LIN {X 0,Y 250.875,Z 1142.399,A -85,B 0,C 180,E1 12020.082,E2 12020.082} C_VEL
LIN {X 0,Y 256.452,Z 1121.884,A -85,B 0,C 180,E1 12017.28,E2 12017.28} C_VEL
LIN {X 0,Y 262.071,Z 1099.557,A -85,B 0,C 180,E1 12014.793,E2 12014.793} C_VEL
LIN {X 0,Y 267.365,Z 1075.91,A -85,B 0,C 180,E1 12012.685,E2 12012.685} C_VEL
LIN {X 0,Y 272.115,Z 1051.396,A -85,B 0,C 180,E1 12010.964,E2 12010.964} C_VEL
LIN {X 0,Y 276.224,Z 1025.533,A -85,B 0,C 180,E1 12009.582,E2 12009.582} C_VEL
LIN {X 0,Y 282.995,Z 970.684,A -85,B 0,C 180,E1 12007.498,E2 12007.498} C_VEL
LIN {X 0,Y 300.587,Z 832.085,A -85,B 0,C 180,E1 12002.78,E2 12002.78} C_VEL
LIN {X 0,Y 288.306,Z 807.074,A -85,B 0,C 180,E1 11999.364,E2 11999.364} C_VEL
LIN {X 0,Y 276.041,Z 783.888,A -85,B 0,C 180,E1 11995.652,E2 11995.652} C_VEL
LIN {X 0,Y 264.408,Z 763.41,A -85,B 0,C 180,E1 11991.784,E2 11991.784} C_VEL
LIN {X 0,Y 253.537,Z 745.664,A -85,B 0,C 180,E1 11987.8,E2 11987.8} C_VEL
LIN {X 0,Y 245.018,Z 732.558,A -85,B 0,C 180,E1 11984.357,E2 11984.357} C_VEL
LIN {X 0,Y 243.38,Z 730.234,A -85,B 0,C 180,E1 11983.667,E2 11983.667} C_VEL
LIN {X 0,Y 242.49,Z 729.861,A -85,B 0,C 180,E1 11983.311,E2 11983.311} C_VEL
LIN {X 0,Y 243.74,Z 731.685,A -85,B 0,C 180,E1 11981.348,E2 11981.348} C_VEL
LIN {X 0,Y 246.278,Z 736.647,A -85,B 0,C 180,E1 11977.233,E2 11977.233} C_VEL
LIN {X 0,Y 248.775,Z 741.662,A -85,B 0,C 180,E1 11973.69,E2 11973.69} C_VEL
LIN {X 0,Y 251.092,Z 746.409,A -85,B 0,C 180,E1 11970.688,E2 11970.688} C_VEL
LIN {X 0,Y 254.649,Z 753.588,A -85,B 0,C 180,E1 11966.627,E2 11966.627} C_VEL
LIN {X 0,Y 258.733,Z 762.816,A -85,B 0,C 180,E1 11962.23,E2 11962.23} C_VEL
LIN {X 0,Y 263.13,Z 773.088,A -85,B 0,C 180,E1 11957.94,E2 11957.94} C_VEL
LIN {X 0,Y 267.756,Z 784.772,A -85,B 0,C 180,E1 11953.685,E2 11953.685} C_VEL
LIN {X 0,Y 272.379,Z 797.535,A -85,B 0,C 180,E1 11949.593,E2 11949.593} C_VEL
LIN {X 0,Y 277.126,Z 811.99,A -85,B 0,C 180,E1 11945.489,E2 11945.489} C_VEL
LIN {X 0,Y 281.607,Z 827.392,A -85,B 0,C 180,E1 11941.593,E2 11941.593} C_VEL
LIN {X 0,Y 283.554,Z 835.371,A -85,B 0,C 180,E1 11939.762,E2 11939.762} C_VEL
LIN {X 0,Y 271.947,Z 876.824,A -85,B 0,C 180,E1 11934.348,E2 11934.348} C_VEL
LIN {X 0,Y 261.07,Z 920.048,A -85,B 0,C 180,E1 11928.508,E2 11928.508} C_VEL
LIN {X 0,Y 258.223,Z 932.884,A -85,B 0,C 180,E1 11926.79,E2 11926.79} C_VEL
LIN {X 0,Y 257.872,Z 942.975,A -85,B 0,C 180,E1 11926.225,E2 11926.225} C_VEL
LIN {X 0,Y 250.822,Z 1001.369,A -85,B 0,C 180,E1 11923.289,E2 11923.289} C_VEL
LIN {X 0,Y 244.667,Z 1051.459,A -85,B 0,C 180,E1 11920.196,E2 11920.196} C_VEL
LIN {X 0,Y 240.696,Z 1089.833,A -85,B 0,C 180,E1 11917.338,E2 11917.338} C_VEL
LIN {X 0,Y 238.457,Z 1107.896,A -85,B 0,C 180,E1 11915.523,E2 11915.523} C_VEL
LIN {X 0,Y 236.095,Z 1124.174,A -85,B 0,C 180,E1 11913.406,E2 11913.406} C_VEL
LIN {X 0,Y 233.562,Z 1140.25,A -85,B 0,C 180,E1 11910.77,E2 11910.77} C_VEL
LIN {X 0,Y 231.041,Z 1155.81,A -85,B 0,C 180,E1 11907.586,E2 11907.586} C_VEL
LIN {X 0,Y 228.852,Z 1169.954,A -85,B 0,C 180,E1 11903.975,E2 11903.975} C_VEL
LIN {X 0,Y 227.359,Z 1181.506,A -85,B 0,C 180,E1 11900.33,E2 11900.33} C_VEL
LIN {X 0,Y 226.431,Z 1192.191,A -85,B 0,C 180,E1 11896.153,E2 11896.153} C_VEL
LIN {X 0,Y 226.295,Z 1201.142,A -85,B 0,C 180,E1 11891.727,E2 11891.727} C_VEL
LIN {X 0,Y 227.021,Z 1207.997,A -85,B 0,C 180,E1 11887.338,E2 11887.338} C_VEL
LIN {X 0,Y 228.861,Z 1213.356,A -85,B 0,C 180,E1 11882.755,E2 11882.755} C_VEL
LIN {X 0,Y 232.16,Z 1217.018,A -85,B 0,C 180,E1 11878.025,E2 11878.025} C_VEL
LIN {X 0,Y 236.961,Z 1218.837,A -85,B 0,C 180,E1 11873.458,E2 11873.458} C_VEL
LIN {X 0,Y 243.636,Z 1218.792,A -85,B 0,C 180,E1 11868.878,E2 11868.878} C_VEL
LIN {X 0,Y 252.162,Z 1216.676,A -85,B 0,C 180,E1 11864.47,E2 11864.47} C_VEL
LIN {X 0,Y 261.202,Z 1213.007,A -85,B 0,C 180,E1 11860.779,E2 11860.779} C_VEL
LIN {X 0,Y 271.771,Z 1207.47,A -85,B 0,C 180,E1 11857.275,E2 11857.275} C_VEL
LIN {X 0,Y 283.551,Z 1200.008,A -85,B 0,C 180,E1 11854.07,E2 11854.07} C_VEL
LIN {X 0,Y 286.866,Z 1197.645,A -85,B 0,C 180,E1 11853.267,E2 11853.267} C_VEL
LIN {X 0,Y 290.92,Z 1194.738,A -85,B 0,C 180,E1 11852.083,E2 11852.083} C_VEL
LIN {X 0,Y 299.595,Z 1187.805,A -85,B 0,C 180,E1 11848.837,E2 11848.837} C_VEL
LIN {X 0,Y 303.94,Z 1184.184,A -85,B 0,C 180,E1 11847.843,E2 11847.843} C_VEL
LIN {X 0,Y 312.8,Z 1176.577,A -85,B 0,C 180,E1 11846.411,E2 11846.411} C_VEL
LIN {X 0,Y 298.241,Z 1190.287,A -85,B 0,C 180,E1 11844.221,E2 11844.221} C_VEL
LIN {X 0,Y 282.111,Z 1204.39,A -85,B 0,C 180,E1 11841.232,E2 11841.232} C_VEL
LIN {X 0,Y 267.332,Z 1216.538,A -85,B 0,C 180,E1 11837.775,E2 11837.775} C_VEL
LIN {X 0,Y 252.966,Z 1227.89,A -85,B 0,C 180,E1 11833.448,E2 11833.448} C_VEL
LIN {X 0,Y 240.286,Z 1237.665,A -85,B 0,C 180,E1 11828.313,E2 11828.313} C_VEL
LIN {X 0,Y 230.902,Z 1244.993,A -85,B 0,C 180,E1 11823.063,E2 11823.063} C_VEL
LIN {X 0,Y 223.215,Z 1251.335,A -85,B 0,C 180,E1 11816.608,E2 11816.608} C_VEL
LIN {X 0,Y 218.765,Z 1255.587,A -85,B 0,C 180,E1 11809.687,E2 11809.687} C_VEL
LIN {X 0,Y 217.644,Z 1257.45,A -85,B 0,C 180,E1 11804.496,E2 11804.496} C_VEL
LIN {X 0,Y 217.156,Z 1265.482,A -85,B 0,C 180,E1 11799.805,E2 11799.805} C_VEL
LIN {X 0,Y 217.229,Z 1272.099,A -85,B 0,C 180,E1 11795.014,E2 11795.014} C_VEL
LIN {X 0,Y 217.292,Z 1276.222,A -85,B 0,C 180,E1 11791.051,E2 11791.051} C_VEL
LIN {X 0,Y 217,Z 1279.073,A -85,B 0,C 180,E1 11787.355,E2 11787.355} C_VEL
LIN {X 0,Y 216.544,Z 1281.409,A -85,B 0,C 180,E1 11782.835,E2 11782.835} C_VEL
LIN {X 0,Y 216.902,Z 1282.929,A -85,B 0,C 180,E1 11776.578,E2 11776.578} C_VEL
LIN {X 0,Y 219.361,Z 1282.777,A -85,B 0,C 180,E1 11770.284,E2 11770.284} C_VEL
LIN {X 0,Y 224.928,Z 1280.78,A -85,B 0,C 180,E1 11763.603,E2 11763.603} C_VEL
LIN {X 0,Y 234.376,Z 1276.835,A -85,B 0,C 180,E1 11756.899,E2 11756.899} C_VEL
LIN {X 0,Y 246.727,Z 1271.422,A -85,B 0,C 180,E1 11751.083,E2 11751.083} C_VEL
LIN {X 0,Y 263.196,Z 1263.992,A -85,B 0,C 180,E1 11745.648,E2 11745.648} C_VEL
LIN {X 0,Y 272.977,Z 1259.532,A -85,B 0,C 180,E1 11743.089,E2 11743.089} C_VEL
LIN {X 0,Y 255.858,Z 1264.797,A -85,B 0,C 180,E1 11738.131,E2 11738.131} C_VEL
LIN {X 0,Y 241.819,Z 1268.371,A -85,B 0,C 180,E1 11732.516,E2 11732.516} C_VEL
LIN {X 0,Y 231.077,Z 1270.191,A -85,B 0,C 180,E1 11726.395,E2 11726.395} C_VEL
LIN {X 0,Y 223.504,Z 1270.13,A -85,B 0,C 180,E1 11719.877,E2 11719.877} C_VEL
LIN {X 0,Y 219.062,Z 1268.343,A -85,B 0,C 180,E1 11713.461,E2 11713.461} C_VEL
LIN {X 0,Y 216.939,Z 1264.947,A -85,B 0,C 180,E1 11707.149,E2 11707.149} C_VEL
LIN {X 0,Y 216.319,Z 1260.682,A -85,B 0,C 180,E1 11701.854,E2 11701.854} C_VEL
LIN {X 0,Y 216.214,Z 1255.219,A -85,B 0,C 180,E1 11696.819,E2 11696.819} C_VEL
LIN {X 0,Y 216.471,Z 1248.644,A -85,B 0,C 180,E1 11692.035,E2 11692.035} C_VEL
LIN {X 0,Y 217.315,Z 1239.961,A -85,B 0,C 180,E1 11686.97,E2 11686.97} C_VEL
LIN {X 0,Y 218.948,Z 1230.048,A -85,B 0,C 180,E1 11682.183,E2 11682.183} C_VEL
LIN {X 0,Y 221.732,Z 1217.438,A -85,B 0,C 180,E1 11677.181,E2 11677.181} C_VEL
LIN {X 0,Y 225.229,Z 1204.04,A -85,B 0,C 180,E1 11672.789,E2 11672.789} C_VEL
LIN {X 0,Y 229.707,Z 1188.379,A -85,B 0,C 180,E1 11668.51,E2 11668.51} C_VEL
LIN {X 0,Y 235.034,Z 1170.475,A -85,B 0,C 180,E1 11664.468,E2 11664.468} C_VEL
LIN {X 0,Y 240.517,Z 1152.019,A -85,B 0,C 180,E1 11661.028,E2 11661.028} C_VEL
LIN {X 0,Y 246.057,Z 1132.723,A -85,B 0,C 180,E1 11658.047,E2 11658.047} C_VEL
LIN {X 0,Y 251.937,Z 1110.749,A -85,B 0,C 180,E1 11655.272,E2 11655.272} C_VEL
LIN {X 0,Y 257.513,Z 1087.985,A -85,B 0,C 180,E1 11652.952,E2 11652.952} C_VEL
LIN {X 0,Y 262.772,Z 1063.42,A -85,B 0,C 180,E1 11650.963,E2 11650.963} C_VEL
LIN {X 0,Y 267.339,Z 1038.17,A -85,B 0,C 180,E1 11649.382,E2 11649.382} C_VEL
LIN {X 0,Y 271.084,Z 1012.485,A -85,B 0,C 180,E1 11648.187,E2 11648.187} C_VEL
LIN {X 0,Y 294.09,Z 834.845,A -85,B 0,C 180,E1 11641.891,E2 11641.891} C_VEL
LIN {X 0,Y 282.266,Z 810.63,A -85,B 0,C 180,E1 11638.485,E2 11638.485} C_VEL
LIN {X 0,Y 269.829,Z 787,A -85,B 0,C 180,E1 11634.582,E2 11634.582} C_VEL
LIN {X 0,Y 258.588,Z 767.172,A -85,B 0,C 180,E1 11630.694,E2 11630.694} C_VEL
LIN {X 0,Y 248.246,Z 750.166,A -85,B 0,C 180,E1 11626.741,E2 11626.741} C_VEL
LIN {X 0,Y 240.071,Z 737.582,A -85,B 0,C 180,E1 11623.307,E2 11623.307} C_VEL
LIN {X 0,Y 238.286,Z 736.957,A -85,B 0,C 180,E1 11622.668,E2 11622.668} C_VEL
LIN {X 0,Y 239.049,Z 738.368,A -85,B 0,C 180,E1 11621.341,E2 11621.341} C_VEL
LIN {X 0,Y 241.442,Z 743.073,A -85,B 0,C 180,E1 11617.379,E2 11617.379} C_VEL
LIN {X 0,Y 243.73,Z 747.729,A -85,B 0,C 180,E1 11614.002,E2 11614.002} C_VEL
LIN {X 0,Y 246.014,Z 752.518,A -85,B 0,C 180,E1 11610.935,E2 11610.935} C_VEL
LIN {X 0,Y 249.344,Z 759.346,A -85,B 0,C 180,E1 11607.015,E2 11607.015} C_VEL
LIN {X 0,Y 253.36,Z 768.616,A -85,B 0,C 180,E1 11602.52,E2 11602.52} C_VEL
LIN {X 0,Y 257.48,Z 778.43,A -85,B 0,C 180,E1 11598.353,E2 11598.353} C_VEL
LIN {X 0,Y 261.961,Z 790.021,A -85,B 0,C 180,E1 11594.052,E2 11594.052} C_VEL
LIN {X 0,Y 266.557,Z 803.069,A -85,B 0,C 180,E1 11589.815,E2 11589.815} C_VEL
LIN {X 0,Y 270.992,Z 816.903,A -85,B 0,C 180,E1 11585.826,E2 11585.826} C_VEL
LIN {X 0,Y 275.393,Z 832.431,A -85,B 0,C 180,E1 11581.84,E2 11581.84} C_VEL
LIN {X 0,Y 276.758,Z 837.922,A -85,B 0,C 180,E1 11580.541,E2 11580.541} C_VEL
LIN {X 0,Y 265.024,Z 878.564,A -85,B 0,C 180,E1 11575.15,E2 11575.15} C_VEL
LIN {X 0,Y 253.698,Z 922.243,A -85,B 0,C 180,E1 11569.142,E2 11569.142} C_VEL
LIN {X 0,Y 251.096,Z 933.637,A -85,B 0,C 180,E1 11567.59,E2 11567.59} C_VEL
LIN {X 0,Y 250.715,Z 943.422,A -85,B 0,C 180,E1 11567.033,E2 11567.033} C_VEL
LIN {X 0,Y 243.82,Z 998.613,A -85,B 0,C 180,E1 11564.177,E2 11564.177} C_VEL
LIN {X 0,Y 237.333,Z 1049.608,A -85,B 0,C 180,E1 11560.958,E2 11560.958} C_VEL
LIN {X 0,Y 232.982,Z 1090.078,A -85,B 0,C 180,E1 11557.852,E2 11557.852} C_VEL
LIN {X 0,Y 230.665,Z 1108.034,A -85,B 0,C 180,E1 11555.971,E2 11555.971} C_VEL
LIN {X 0,Y 228.111,Z 1125.131,A -85,B 0,C 180,E1 11553.661,E2 11553.661} C_VEL
LIN {X 0,Y 225.535,Z 1141.103,A -85,B 0,C 180,E1 11550.949,E2 11550.949} C_VEL
LIN {X 0,Y 222.971,Z 1156.657,A -85,B 0,C 180,E1 11547.654,E2 11547.654} C_VEL
LIN {X 0,Y 220.964,Z 1169.36,A -85,B 0,C 180,E1 11544.317,E2 11544.317} C_VEL
LIN {X 0,Y 219.402,Z 1181.16,A -85,B 0,C 180,E1 11540.543,E2 11540.543} C_VEL
LIN {X 0,Y 218.435,Z 1192.08,A -85,B 0,C 180,E1 11536.214,E2 11536.214} C_VEL
LIN {X 0,Y 218.282,Z 1200.761,A -85,B 0,C 180,E1 11531.896,E2 11531.896} C_VEL
LIN {X 0,Y 219.076,Z 1208.382,A -85,B 0,C 180,E1 11527.079,E2 11527.079} C_VEL
LIN {X 0,Y 221.172,Z 1214.172,A -85,B 0,C 180,E1 11522.073,E2 11522.073} C_VEL
LIN {X 0,Y 224.512,Z 1217.875,A -85,B 0,C 180,E1 11517.447,E2 11517.447} C_VEL
LIN {X 0,Y 229.955,Z 1220.047,A -85,B 0,C 180,E1 11512.442,E2 11512.442} C_VEL
LIN {X 0,Y 237.355,Z 1220.141,A -85,B 0,C 180,E1 11507.594,E2 11507.594} C_VEL
LIN {X 0,Y 246.17,Z 1218.264,A -85,B 0,C 180,E1 11503.239,E2 11503.239} C_VEL
LIN {X 0,Y 255.969,Z 1214.718,A -85,B 0,C 180,E1 11499.417,E2 11499.417} C_VEL
LIN {X 0,Y 267.678,Z 1209.064,A -85,B 0,C 180,E1 11495.739,E2 11495.739} C_VEL
LIN {X 0,Y 280.71,Z 1201.313,A -85,B 0,C 180,E1 11492.415,E2 11492.415} C_VEL
LIN {X 0,Y 294.866,Z 1191.373,A -85,B 0,C 180,E1 11489.458,E2 11489.458} C_VEL
LIN {X 0,Y 303.94,Z 1184.184,A -85,B 0,C 180,E1 11487.843,E2 11487.843} C_VEL
LIN {X 0,Y 304.402,Z 1183.842,A -85,B 0,C 180,E1 11487.518,E2 11487.518} C_VEL
LIN {X 0,Y 303.522,Z 1184.706,A -85,B 0,C 180,E1 11486.987,E2 11486.987} C_VEL
LIN {X 0,Y 300.875,Z 1187.091,A -85,B 0,C 180,E1 11486.354,E2 11486.354} C_VEL
LIN {X 0,Y 290.176,Z 1196.083,A -85,B 0,C 180,E1 11484.823,E2 11484.823} C_VEL
LIN {X 0,Y 274.447,Z 1208.597,A -85,B 0,C 180,E1 11481.896,E2 11481.896} C_VEL
LIN {X 0,Y 257.544,Z 1221.216,A -85,B 0,C 180,E1 11477.857,E2 11477.857} C_VEL
LIN {X 0,Y 243.247,Z 1231.39,A -85,B 0,C 180,E1 11473.346,E2 11473.346} C_VEL
LIN {X 0,Y 230.704,Z 1240.16,A -85,B 0,C 180,E1 11467.979,E2 11467.979} C_VEL
LIN {X 0,Y 220.55,Z 1247.296,A -85,B 0,C 180,E1 11461.724,E2 11461.724} C_VEL
LIN {X 0,Y 213.847,Z 1252.248,A -85,B 0,C 180,E1 11455.177,E2 11455.177} C_VEL
LIN {X 0,Y 210.379,Z 1255.245,A -85,B 0,C 180,E1 11448.564,E2 11448.564} C_VEL
LIN {X 0,Y 209.727,Z 1256.284,A -85,B 0,C 180,E1 11444.505,E2 11444.505} C_VEL
LIN {X 0,Y 209.246,Z 1264.452,A -85,B 0,C 180,E1 11439.624,E2 11439.624} C_VEL
LIN {X 0,Y 209.334,Z 1270.834,A -85,B 0,C 180,E1 11434.928,E2 11434.928} C_VEL
LIN {X 0,Y 209.389,Z 1275.325,A -85,B 0,C 180,E1 11430.543,E2 11430.543} C_VEL
LIN {X 0,Y 208.992,Z 1278.362,A -85,B 0,C 180,E1 11426.43,E2 11426.43} C_VEL
LIN {X 0,Y 208.563,Z 1280.777,A -85,B 0,C 180,E1 11421.449,E2 11421.449} C_VEL
LIN {X 0,Y 209.408,Z 1282.29,A -85,B 0,C 180,E1 11414.693,E2 11414.693} C_VEL
LIN {X 0,Y 212.805,Z 1282.066,A -85,B 0,C 180,E1 11407.917,E2 11407.917} C_VEL
LIN {X 0,Y 219.493,Z 1280.04,A -85,B 0,C 180,E1 11401.123,E2 11401.123} C_VEL
LIN {X 0,Y 230.233,Z 1276.193,A -85,B 0,C 180,E1 11394.408,E2 11394.408} C_VEL
LIN {X 0,Y 244.372,Z 1270.712,A -85,B 0,C 180,E1 11388.479,E2 11388.479} C_VEL
LIN {X 0,Y 262.804,Z 1263.261,A -85,B 0,C 180,E1 11383.046,E2 11383.046} C_VEL
LIN {X 0,Y 245.305,Z 1267.667,A -85,B 0,C 180,E1 11377.692,E2 11377.692} C_VEL
LIN {X 0,Y 231.563,Z 1270.259,A -85,B 0,C 180,E1 11371.789,E2 11371.789} C_VEL
LIN {X 0,Y 220.986,Z 1271.089,A -85,B 0,C 180,E1 11365.171,E2 11365.171} C_VEL
LIN {X 0,Y 214.164,Z 1270.054,A -85,B 0,C 180,E1 11358.511,E2 11358.511} C_VEL
LIN {X 0,Y 210.276,Z 1267.369,A -85,B 0,C 180,E1 11351.799,E2 11351.799} C_VEL
LIN {X 0,Y 208.698,Z 1263.534,A -85,B 0,C 180,E1 11345.774,E2 11345.774} C_VEL
LIN {X 0,Y 208.282,Z 1258.51,A -85,B 0,C 180,E1 11340.275,E2 11340.275} C_VEL
LIN {X 0,Y 208.282,Z 1252.371,A -85,B 0,C 180,E1 11335.043,E2 11335.043} C_VEL
LIN {X 0,Y 208.723,Z 1244.955,A -85,B 0,C 180,E1 11330.069,E2 11330.069} C_VEL
LIN {X 0,Y 209.936,Z 1235.41,A -85,B 0,C 180,E1 11324.814,E2 11324.814} C_VEL
LIN {X 0,Y 212.097,Z 1224.263,A -85,B 0,C 180,E1 11319.751,E2 11319.751} C_VEL
LIN {X 0,Y 215.417,Z 1210.767,A -85,B 0,C 180,E1 11314.72,E2 11314.72} C_VEL
LIN {X 0,Y 219.505,Z 1196.172,A -85,B 0,C 180,E1 11310.23,E2 11310.23} C_VEL
LIN {X 0,Y 224.292,Z 1180.211,A -85,B 0,C 180,E1 11306.134,E2 11306.134} C_VEL
LIN {X 0,Y 229.785,Z 1162.249,A -85,B 0,C 180,E1 11302.311,E2 11302.311} C_VEL
LIN {X 0,Y 235.46,Z 1143.367,A -85,B 0,C 180,E1 11298.997,E2 11298.997} C_VEL
LIN {X 0,Y 241.296,Z 1122.952,A -85,B 0,C 180,E1 11296.045,E2 11296.045} C_VEL
LIN {X 0,Y 247.431,Z 1099.738,A -85,B 0,C 180,E1 11293.331,E2 11293.331} C_VEL
LIN {X 0,Y 252.947,Z 1076.373,A -85,B 0,C 180,E1 11291.145,E2 11291.145} C_VEL
LIN {X 0,Y 257.953,Z 1051.871,A -85,B 0,C 180,E1 11289.347,E2 11289.347} C_VEL
LIN {X 0,Y 262.269,Z 1026.141,A -85,B 0,C 180,E1 11287.911,E2 11287.911} C_VEL
LIN {X 0,Y 269.578,Z 970.436,A -85,B 0,C 180,E1 11285.69,E2 11285.69} C_VEL
LIN {X 0,Y 287.556,Z 837.478,A -85,B 0,C 180,E1 11280.975,E2 11280.975} C_VEL
LIN {X 0,Y 275.939,Z 813.614,A -85,B 0,C 180,E1 11277.49,E2 11277.49} C_VEL
LIN {X 0,Y 263.65,Z 790.111,A -85,B 0,C 180,E1 11273.469,E2 11273.469} C_VEL
LIN {X 0,Y 252.718,Z 770.807,A -85,B 0,C 180,E1 11269.535,E2 11269.535} C_VEL
LIN {X 0,Y 242.447,Z 753.791,A -85,B 0,C 180,E1 11265.43,E2 11265.43} C_VEL
LIN {X 0,Y 236.695,Z 744.966,A -85,B 0,C 180,E1 11262.941,E2 11262.941} C_VEL
LIN {X 0,Y 234.073,Z 744.17,A -85,B 0,C 180,E1 11261.978,E2 11261.978} C_VEL
LIN {X 0,Y 236.45,Z 749.097,A -85,B 0,C 180,E1 11257.78,E2 11257.78} C_VEL
LIN {X 0,Y 238.834,Z 754.179,A -85,B 0,C 180,E1 11254.084,E2 11254.084} C_VEL
LIN {X 0,Y 241.02,Z 758.781,A -85,B 0,C 180,E1 11251.112,E2 11251.112} C_VEL
LIN {X 0,Y 244.232,Z 765.571,A -85,B 0,C 180,E1 11247.187,E2 11247.187} C_VEL
LIN {X 0,Y 248.216,Z 774.921,A -85,B 0,C 180,E1 11242.597,E2 11242.597} C_VEL
LIN {X 0,Y 252.265,Z 784.901,A -85,B 0,C 180,E1 11238.341,E2 11238.341} C_VEL
LIN {X 0,Y 256.695,Z 796.682,A -85,B 0,C 180,E1 11233.948,E2 11233.948} C_VEL
LIN {X 0,Y 261.216,Z 809.977,A -85,B 0,C 180,E1 11229.618,E2 11229.618} C_VEL
LIN {X 0,Y 265.549,Z 824.178,A -85,B 0,C 180,E1 11225.535,E2 11225.535} C_VEL
LIN {X 0,Y 269.933,Z 840.364,A -85,B 0,C 180,E1 11221.391,E2 11221.391} C_VEL
LIN {X 0,Y 259.912,Z 874.128,A -85,B 0,C 180,E1 11216.834,E2 11216.834} C_VEL
LIN {X 0,Y 248.193,Z 917.054,A -85,B 0,C 180,E1 11210.853,E2 11210.853} C_VEL
LIN {X 0,Y 243.991,Z 934.422,A -85,B 0,C 180,E1 11208.422,E2 11208.422} C_VEL
LIN {X 0,Y 243.553,Z 943.881,A -85,B 0,C 180,E1 11207.863,E2 11207.863} C_VEL
LIN {X 0,Y 236.297,Z 1000.213,A -85,B 0,C 180,E1 11204.857,E2 11204.857} C_VEL
LIN {X 0,Y 229.721,Z 1050.451,A -85,B 0,C 180,E1 11201.572,E2 11201.572} C_VEL
LIN {X 0,Y 225.225,Z 1090.329,A -85,B 0,C 180,E1 11198.347,E2 11198.347} C_VEL
LIN {X 0,Y 222.934,Z 1107.714,A -85,B 0,C 180,E1 11196.486,E2 11196.486} C_VEL
LIN {X 0,Y 220.292,Z 1125.073,A -85,B 0,C 180,E1 11194.095,E2 11194.095} C_VEL
LIN {X 0,Y 217.626,Z 1141.263,A -85,B 0,C 180,E1 11191.278,E2 11191.278} C_VEL
LIN {X 0,Y 215.058,Z 1156.417,A -85,B 0,C 180,E1 11187.956,E2 11187.956} C_VEL
LIN {X 0,Y 212.922,Z 1169.739,A -85,B 0,C 180,E1 11184.363,E2 11184.363} C_VEL
LIN {X 0,Y 211.276,Z 1182.286,A -85,B 0,C 180,E1 11180.211,E2 11180.211} C_VEL
LIN {X 0,Y 210.376,Z 1193.092,A -85,B 0,C 180,E1 11175.719,E2 11175.719} C_VEL
LIN {X 0,Y 210.326,Z 1201.795,A -85,B 0,C 180,E1 11171.24,E2 11171.24} C_VEL
LIN {X 0,Y 211.297,Z 1209.383,A -85,B 0,C 180,E1 11166.248,E2 11166.248} C_VEL
LIN {X 0,Y 213.513,Z 1214.978,A -85,B 0,C 180,E1 11161.342,E2 11161.342} C_VEL
LIN {X 0,Y 217.425,Z 1219.045,A -85,B 0,C 180,E1 11156.247,E2 11156.247} C_VEL
LIN {X 0,Y 223.531,Z 1221.324,A -85,B 0,C 180,E1 11150.993,E2 11150.993} C_VEL
LIN {X 0,Y 231.641,Z 1221.471,A -85,B 0,C 180,E1 11146.011,E2 11146.011} C_VEL
LIN {X 0,Y 241.081,Z 1219.663,A -85,B 0,C 180,E1 11141.626,E2 11141.626} C_VEL
LIN {X 0,Y 251.479,Z 1216.217,A -85,B 0,C 180,E1 11137.807,E2 11137.807} C_VEL
LIN {X 0,Y 263.812,Z 1210.705,A -85,B 0,C 180,E1 11134.159,E2 11134.159} C_VEL
LIN {X 0,Y 277.455,Z 1203.147,A -85,B 0,C 180,E1 11130.888,E2 11130.888} C_VEL
LIN {X 0,Y 291.535,Z 1193.926,A -85,B 0,C 180,E1 11128.117,E2 11128.117} C_VEL
LIN {X 0,Y 300.971,Z 1186.973,A -85,B 0,C 180,E1 11126.493,E2 11126.493} C_VEL
LIN {X 0,Y 290.176,Z 1196.083,A -85,B 0,C 180,E1 11124.823,E2 11124.823} C_VEL
LIN {X 0,Y 284.673,Z 1200.4,A -85,B 0,C 180,E1 11124.132,E2 11124.132} C_VEL
LIN {X 0,Y 268.972,Z 1211.132,A -85,B 0,C 180,E1 11122.772,E2 11122.772} C_VEL
LIN {X 0,Y 263.532,Z 1214.717,A -85,B 0,C 180,E1 11121.902,E2 11121.902} C_VEL
LIN {X 0,Y 247.566,Z 1225.403,A -85,B 0,C 180,E1 11117.898,E2 11117.898} C_VEL
LIN {X 0,Y 232.974,Z 1234.797,A -85,B 0,C 180,E1 11113.026,E2 11113.026} C_VEL
LIN {X 0,Y 219.821,Z 1242.974,A -85,B 0,C 180,E1 11106.895,E2 11106.895} C_VEL
LIN {X 0,Y 210.97,Z 1248.517,A -85,B 0,C 180,E1 11100.783,E2 11100.783} C_VEL
LIN {X 0,Y 204.661,Z 1252.666,A -85,B 0,C 180,E1 11093.612,E2 11093.612} C_VEL
LIN {X 0,Y 201.928,Z 1254.738,A -85,B 0,C 180,E1 11086.095,E2 11086.095} C_VEL
LIN {X 0,Y 201.816,Z 1255.095,A -85,B 0,C 180,E1 11084.485,E2 11084.485} C_VEL
LIN {X 0,Y 201.345,Z 1263.795,A -85,B 0,C 180,E1 11079.14,E2 11079.14} C_VEL
LIN {X 0,Y 201.471,Z 1269.79,A -85,B 0,C 180,E1 11074.551,E2 11074.551} C_VEL
LIN {X 0,Y 201.496,Z 1274.157,A -85,B 0,C 180,E1 11070.28,E2 11070.28} C_VEL
LIN {X 0,Y 201.018,Z 1277.45,A -85,B 0,C 180,E1 11065.717,E2 11065.717} C_VEL
LIN {X 0,Y 200.643,Z 1279.895,A -85,B 0,C 180,E1 11060.531,E2 11060.531} C_VEL
LIN {X 0,Y 201.674,Z 1281.549,A -85,B 0,C 180,E1 11053.877,E2 11053.877} C_VEL
LIN {X 0,Y 205.503,Z 1281.497,A -85,B 0,C 180,E1 11046.786,E2 11046.786} C_VEL
LIN {X 0,Y 213.437,Z 1279.648,A -85,B 0,C 180,E1 11039.29,E2 11039.29} C_VEL
LIN {X 0,Y 225.125,Z 1276.088,A -85,B 0,C 180,E1 11032.516,E2 11032.516} C_VEL
LIN {X 0,Y 240.801,Z 1270.71,A -85,B 0,C 180,E1 11026.423,E2 11026.423} C_VEL
LIN {X 0,Y 252.564,Z 1266.513,A -85,B 0,C 180,E1 11022.995,E2 11022.995} C_VEL
LIN {X 0,Y 235.821,Z 1269.863,A -85,B 0,C 180,E1 11017.631,E2 11017.631} C_VEL
LIN {X 0,Y 221.748,Z 1271.626,A -85,B 0,C 180,E1 11011.235,E2 11011.235} C_VEL
LIN {X 0,Y 211.809,Z 1271.499,A -85,B 0,C 180,E1 11004.546,E2 11004.546} C_VEL
LIN {X 0,Y 205.314,Z 1269.704,A -85,B 0,C 180,E1 10997.574,E2 10997.574} C_VEL
LIN {X 0,Y 201.892,Z 1266.47,A -85,B 0,C 180,E1 10990.848,E2 10990.848} C_VEL
LIN {X 0,Y 200.592,Z 1262.14,A -85,B 0,C 180,E1 10984.861,E2 10984.861} C_VEL
LIN {X 0,Y 200.282,Z 1256.958,A -85,B 0,C 180,E1 10979.428,E2 10979.428} C_VEL
LIN {X 0,Y 200.349,Z 1250.602,A -85,B 0,C 180,E1 10974.271,E2 10974.271} C_VEL
LIN {X 0,Y 200.945,Z 1242.319,A -85,B 0,C 180,E1 10968.81,E2 10968.81} C_VEL
LIN {X 0,Y 202.327,Z 1232.699,A -85,B 0,C 180,E1 10963.639,E2 10963.639} C_VEL
LIN {X 0,Y 204.726,Z 1221.189,A -85,B 0,C 180,E1 10958.512,E2 10958.512} C_VEL
LIN {X 0,Y 208.261,Z 1207.567,A -85,B 0,C 180,E1 10953.48,E2 10953.48} C_VEL
LIN {X 0,Y 212.726,Z 1192.327,A -85,B 0,C 180,E1 10948.817,E2 10948.817} C_VEL
LIN {X 0,Y 217.993,Z 1175.35,A -85,B 0,C 180,E1 10944.533,E2 10944.533} C_VEL
LIN {X 0,Y 224.023,Z 1156.022,A -85,B 0,C 180,E1 10940.552,E2 10940.552} C_VEL
LIN {X 0,Y 230.365,Z 1135.064,A -85,B 0,C 180,E1 10937.042,E2 10937.042} C_VEL
LIN {X 0,Y 236.589,Z 1113.156,A -85,B 0,C 180,E1 10934.072,E2 10934.072} C_VEL
LIN {X 0,Y 242.481,Z 1090.438,A -85,B 0,C 180,E1 10931.601,E2 10931.601} C_VEL
LIN {X 0,Y 247.804,Z 1067.203,A -85,B 0,C 180,E1 10929.584,E2 10929.584} C_VEL
LIN {X 0,Y 252.415,Z 1043.649,A -85,B 0,C 180,E1 10927.973,E2 10927.973} C_VEL
LIN {X 0,Y 256.419,Z 1019.079,A -85,B 0,C 180,E1 10926.696,E2 10926.696} C_VEL
LIN {X 0,Y 281.091,Z 840.162,A -85,B 0,C 180,E1 10920.021,E2 10920.021} C_VEL
LIN {X 0,Y 269.473,Z 816.247,A -85,B 0,C 180,E1 10916.413,E2 10916.413} C_VEL
LIN {X 0,Y 258.059,Z 794.351,A -85,B 0,C 180,E1 10912.529,E2 10912.529} C_VEL
LIN {X 0,Y 247.844,Z 776.099,A -85,B 0,C 180,E1 10908.71,E2 10908.71} C_VEL
LIN {X 0,Y 237.803,Z 759.275,A -85,B 0,C 180,E1 10904.554,E2 10904.554} C_VEL
LIN {X 0,Y 233.464,Z 752.341,A -85,B 0,C 180,E1 10902.62,E2 10902.62} C_VEL
LIN {X 0,Y 229.632,Z 751.67,A -85,B 0,C 180,E1 10901.303,E2 10901.303} C_VEL
LIN {X 0,Y 231.584,Z 755.482,A -85,B 0,C 180,E1 10897.945,E2 10897.945} C_VEL
LIN {X 0,Y 233.818,Z 760.259,A -85,B 0,C 180,E1 10894.418,E2 10894.418} C_VEL
LIN {X 0,Y 236.088,Z 765.171,A -85,B 0,C 180,E1 10891.217,E2 10891.217} C_VEL
LIN {X 0,Y 239.088,Z 771.77,A -85,B 0,C 180,E1 10887.367,E2 10887.367} C_VEL
LIN {X 0,Y 242.835,Z 780.698,A -85,B 0,C 180,E1 10882.908,E2 10882.908} C_VEL
LIN {X 0,Y 246.812,Z 790.76,A -85,B 0,C 180,E1 10878.554,E2 10878.554} C_VEL
LIN {X 0,Y 251.171,Z 802.717,A -85,B 0,C 180,E1 10874.06,E2 10874.06} C_VEL
LIN {X 0,Y 255.599,Z 816.233,A -85,B 0,C 180,E1 10869.629,E2 10869.629} C_VEL
LIN {X 0,Y 259.616,Z 829.878,A -85,B 0,C 180,E1 10865.667,E2 10865.667} C_VEL
LIN {X 0,Y 263.107,Z 843.455,A -85,B 0,C 180,E1 10862.136,E2 10862.136} C_VEL
LIN {X 0,Y 250.235,Z 885.628,A -85,B 0,C 180,E1 10856.358,E2 10856.358} C_VEL
LIN {X 0,Y 238.341,Z 928.969,A -85,B 0,C 180,E1 10850.15,E2 10850.15} C_VEL
LIN {X 0,Y 236.905,Z 935.171,A -85,B 0,C 180,E1 10849.288,E2 10849.288} C_VEL
LIN {X 0,Y 236.421,Z 944.334,A -85,B 0,C 180,E1 10848.734,E2 10848.734} C_VEL
LIN {X 0,Y 229.043,Z 1000.065,A -85,B 0,C 180,E1 10845.687,E2 10845.687} C_VEL
LIN {X 0,Y 222.959,Z 1044.411,A -85,B 0,C 180,E1 10842.711,E2 10842.711} C_VEL
LIN {X 0,Y 217.798,Z 1087.971,A -85,B 0,C 180,E1 10839.124,E2 10839.124} C_VEL
LIN {X 0,Y 215.334,Z 1106.647,A -85,B 0,C 180,E1 10837.132,E2 10837.132} C_VEL
LIN {X 0,Y 212.508,Z 1124.847,A -85,B 0,C 180,E1 10834.58,E2 10834.58} C_VEL
LIN {X 0,Y 209.61,Z 1141.871,A -85,B 0,C 180,E1 10831.49,E2 10831.49} C_VEL
LIN {X 0,Y 207.027,Z 1156.851,A -85,B 0,C 180,E1 10828.093,E2 10828.093} C_VEL
LIN {X 0,Y 204.924,Z 1169.815,A -85,B 0,C 180,E1 10824.503,E2 10824.503} C_VEL
LIN {X 0,Y 203.188,Z 1182.947,A -85,B 0,C 180,E1 10819.977,E2 10819.977} C_VEL
LIN {X 0,Y 202.352,Z 1193.48,A -85,B 0,C 180,E1 10815.476,E2 10815.476} C_VEL
LIN {X 0,Y 202.362,Z 1202.285,A -85,B 0,C 180,E1 10810.822,E2 10810.822} C_VEL
LIN {X 0,Y 203.462,Z 1209.998,A -85,B 0,C 180,E1 10805.641,E2 10805.641} C_VEL
LIN {X 0,Y 205.966,Z 1215.865,A -85,B 0,C 180,E1 10800.433,E2 10800.433} C_VEL
LIN {X 0,Y 210.318,Z 1220.13,A -85,B 0,C 180,E1 10795.091,E2 10795.091} C_VEL
LIN {X 0,Y 216.626,Z 1222.465,A -85,B 0,C 180,E1 10789.898,E2 10789.898} C_VEL
LIN {X 0,Y 224.335,Z 1222.921,A -85,B 0,C 180,E1 10785.267,E2 10785.267} C_VEL
LIN {X 0,Y 234.077,Z 1221.617,A -85,B 0,C 180,E1 10780.797,E2 10780.797} C_VEL
LIN {X 0,Y 246.008,Z 1218.218,A -85,B 0,C 180,E1 10776.527,E2 10776.527} C_VEL
LIN {X 0,Y 259.512,Z 1212.736,A -85,B 0,C 180,E1 10772.709,E2 10772.709} C_VEL
LIN {X 0,Y 274.171,Z 1205.218,A -85,B 0,C 180,E1 10769.386,E2 10769.386} C_VEL
LIN {X 0,Y 289.137,Z 1196.045,A -85,B 0,C 180,E1 10766.586,E2 10766.586} C_VEL
LIN {X 0,Y 271.914,Z 1208.801,A -85,B 0,C 180,E1 10763.634,E2 10763.634} C_VEL
LIN {X 0,Y 263.532,Z 1214.717,A -85,B 0,C 180,E1 10761.902,E2 10761.902} C_VEL
LIN {X 0,Y 258.06,Z 1218.232,A -85,B 0,C 180,E1 10760.961,E2 10760.961} C_VEL
LIN {X 0,Y 242.156,Z 1226.669,A -85,B 0,C 180,E1 10758.908,E2 10758.908} C_VEL
LIN {X 0,Y 236.895,Z 1229.467,A -85,B 0,C 180,E1 10757.737,E2 10757.737} C_VEL
LIN {X 0,Y 222.058,Z 1237.932,A -85,B 0,C 180,E1 10752.399,E2 10752.399} C_VEL
LIN {X 0,Y 210.308,Z 1244.433,A -85,B 0,C 180,E1 10746.458,E2 10746.458} C_VEL
LIN {X 0,Y 200.909,Z 1249.586,A -85,B 0,C 180,E1 10739.186,E2 10739.186} C_VEL
LIN {X 0,Y 195.69,Z 1252.479,A -85,B 0,C 180,E1 10731.896,E2 10731.896} C_VEL
LIN {X 0,Y 193.952,Z 1253.559,A -85,B 0,C 180,E1 10724.628,E2 10724.628} C_VEL
LIN {X 0,Y 193.458,Z 1262.659,A -85,B 0,C 180,E1 10718.916,E2 10718.916} C_VEL
LIN {X 0,Y 193.606,Z 1268.364,A -85,B 0,C 180,E1 10714.439,E2 10714.439} C_VEL
LIN {X 0,Y 193.647,Z 1272.574,A -85,B 0,C 180,E1 10710.292,E2 10710.292} C_VEL
LIN {X 0,Y 193.167,Z 1275.913,A -85,B 0,C 180,E1 10705.84,E2 10705.84} C_VEL
LIN {X 0,Y 192.75,Z 1278.885,A -85,B 0,C 180,E1 10699.837,E2 10699.837} C_VEL
LIN {X 0,Y 194.026,Z 1280.651,A -85,B 0,C 180,E1 10692.914,E2 10692.914} C_VEL
LIN {X 0,Y 198.767,Z 1280.866,A -85,B 0,C 180,E1 10685,E2 10685} C_VEL
LIN {X 0,Y 207.299,Z 1279.357,A -85,B 0,C 180,E1 10677.576,E2 10677.576} C_VEL
LIN {X 0,Y 220.287,Z 1275.913,A -85,B 0,C 180,E1 10670.542,E2 10670.542} C_VEL
LIN {X 0,Y 237.581,Z 1270.777,A -85,B 0,C 180,E1 10664.315,E2 10664.315} C_VEL
LIN {X 0,Y 242.236,Z 1269.297,A -85,B 0,C 180,E1 10662.928,E2 10662.928} C_VEL
LIN {X 0,Y 225.238,Z 1271.773,A -85,B 0,C 180,E1 10657.138,E2 10657.138} C_VEL
LIN {X 0,Y 211.933,Z 1272.498,A -85,B 0,C 180,E1 10650.633,E2 10650.633} C_VEL
LIN {X 0,Y 202.358,Z 1271.51,A -85,B 0,C 180,E1 10643.593,E2 10643.593} C_VEL
LIN {X 0,Y 196.156,Z 1268.742,A -85,B 0,C 180,E1 10635.978,E2 10635.978} C_VEL
LIN {X 0,Y 193.317,Z 1264.618,A -85,B 0,C 180,E1 10628.9,E2 10628.9} C_VEL
LIN {X 0,Y 192.432,Z 1259.443,A -85,B 0,C 180,E1 10622.68,E2 10622.68} C_VEL
LIN {X 0,Y 192.29,Z 1253.783,A -85,B 0,C 180,E1 10617.318,E2 10617.318} C_VEL
LIN {X 0,Y 192.559,Z 1246.553,A -85,B 0,C 180,E1 10611.94,E2 10611.94} C_VEL
LIN {X 0,Y 193.445,Z 1237.833,A -85,B 0,C 180,E1 10606.55,E2 10606.55} C_VEL
LIN {X 0,Y 195.299,Z 1227.235,A -85,B 0,C 180,E1 10601.183,E2 10601.183} C_VEL
LIN {X 0,Y 198.295,Z 1214.64,A -85,B 0,C 180,E1 10595.886,E2 10595.886} C_VEL
LIN {X 0,Y 202.225,Z 1200.739,A -85,B 0,C 180,E1 10591.016,E2 10591.016} C_VEL
LIN {X 0,Y 207.109,Z 1184.959,A -85,B 0,C 180,E1 10586.441,E2 10586.441} C_VEL
LIN {X 0,Y 213.023,Z 1166.462,A -85,B 0,C 180,E1 10582.056,E2 10582.056} C_VEL
LIN {X 0,Y 219.26,Z 1146.762,A -85,B 0,C 180,E1 10578.256,E2 10578.256} C_VEL
LIN {X 0,Y 225.553,Z 1125.973,A -85,B 0,C 180,E1 10575.002,E2 10575.002} C_VEL
LIN {X 0,Y 231.651,Z 1104.265,A -85,B 0,C 180,E1 10572.246,E2 10572.246} C_VEL
LIN {X 0,Y 237.38,Z 1081.78,A -85,B 0,C 180,E1 10569.948,E2 10569.948} C_VEL
LIN {X 0,Y 242.551,Z 1058.604,A -85,B 0,C 180,E1 10568.059,E2 10568.059} C_VEL
LIN {X 0,Y 247.301,Z 1033.431,A -85,B 0,C 180,E1 10566.472,E2 10566.472} C_VEL
LIN {X 0,Y 251.618,Z 1004.472,A -85,B 0,C 180,E1 10565.135,E2 10565.135} C_VEL
LIN {X 0,Y 274.555,Z 842.783,A -85,B 0,C 180,E1 10559.034,E2 10559.034} C_VEL
LIN {X 0,Y 263.188,Z 819.166,A -85,B 0,C 180,E1 10555.336,E2 10555.336} C_VEL
LIN {X 0,Y 251.761,Z 797.137,A -85,B 0,C 180,E1 10551.282,E2 10551.282} C_VEL
LIN {X 0,Y 241.362,Z 778.543,A -85,B 0,C 180,E1 10547.202,E2 10547.202} C_VEL
LIN {X 0,Y 231.658,Z 762.272,A -85,B 0,C 180,E1 10542.973,E2 10542.973} C_VEL
LIN {X 0,Y 230.037,Z 759.85,A -85,B 0,C 180,E1 10542.237,E2 10542.237} C_VEL
LIN {X 0,Y 225.313,Z 759.123,A -85,B 0,C 180,E1 10540.551,E2 10540.551} C_VEL
LIN {X 0,Y 226.749,Z 761.885,A -85,B 0,C 180,E1 10538.115,E2 10538.115} C_VEL
LIN {X 0,Y 228.815,Z 766.343,A -85,B 0,C 180,E1 10534.766,E2 10534.766} C_VEL
LIN {X 0,Y 231.047,Z 771.364,A -85,B 0,C 180,E1 10531.42,E2 10531.42} C_VEL
LIN {X 0,Y 233.932,Z 777.943,A -85,B 0,C 180,E1 10527.554,E2 10527.554} C_VEL
LIN {X 0,Y 237.667,Z 786.959,A -85,B 0,C 180,E1 10522.996,E2 10522.996} C_VEL
LIN {X 0,Y 241.778,Z 797.766,A -85,B 0,C 180,E1 10518.312,E2 10518.312} C_VEL
LIN {X 0,Y 245.84,Z 809.39,A -85,B 0,C 180,E1 10513.948,E2 10513.948} C_VEL
LIN {X 0,Y 249.983,Z 822.466,A -85,B 0,C 180,E1 10509.64,E2 10509.64} C_VEL
LIN {X 0,Y 253.892,Z 836.404,A -85,B 0,C 180,E1 10505.578,E2 10505.578} C_VEL
LIN {X 0,Y 256.287,Z 846.339,A -85,B 0,C 180,E1 10502.97,E2 10502.97} C_VEL
LIN {X 0,Y 243.048,Z 888.386,A -85,B 0,C 180,E1 10497.113,E2 10497.113} C_VEL
LIN {X 0,Y 230.886,Z 931.433,A -85,B 0,C 180,E1 10490.823,E2 10490.823} C_VEL
LIN {X 0,Y 229.862,Z 936.03,A -85,B 0,C 180,E1 10490.196,E2 10490.196} C_VEL
LIN {X 0,Y 229.338,Z 944.839,A -85,B 0,C 180,E1 10489.655,E2 10489.655} C_VEL
LIN {X 0,Y 222.42,Z 995.423,A -85,B 0,C 180,E1 10486.824,E2 10486.824} C_VEL
LIN {X 0,Y 215.55,Z 1043.799,A -85,B 0,C 180,E1 10483.493,E2 10483.493} C_VEL
LIN {X 0,Y 210.1,Z 1088.141,A -85,B 0,C 180,E1 10479.711,E2 10479.711} C_VEL
LIN {X 0,Y 207.626,Z 1106.308,A -85,B 0,C 180,E1 10477.706,E2 10477.706} C_VEL
LIN {X 0,Y 204.822,Z 1123.837,A -85,B 0,C 180,E1 10475.173,E2 10475.173} C_VEL
LIN {X 0,Y 202.098,Z 1139.632,A -85,B 0,C 180,E1 10472.299,E2 10472.299} C_VEL
LIN {X 0,Y 199.362,Z 1155.168,A -85,B 0,C 180,E1 10468.783,E2 10468.783} C_VEL
LIN {X 0,Y 196.911,Z 1169.848,A -85,B 0,C 180,E1 10464.607,E2 10464.607} C_VEL
LIN {X 0,Y 195.286,Z 1181.924,A -85,B 0,C 180,E1 10460.376,E2 10460.376} C_VEL
LIN {X 0,Y 194.388,Z 1192.55,A -85,B 0,C 180,E1 10455.82,E2 10455.82} C_VEL
LIN {X 0,Y 194.376,Z 1202.195,A -85,B 0,C 180,E1 10450.672,E2 10450.672} C_VEL
LIN {X 0,Y 195.447,Z 1209.793,A -85,B 0,C 180,E1 10445.578,E2 10445.578} C_VEL
LIN {X 0,Y 198.119,Z 1216.207,A -85,B 0,C 180,E1 10440,E2 10440} C_VEL
LIN {X 0,Y 202.512,Z 1220.659,A -85,B 0,C 180,E1 10434.617,E2 10434.617} C_VEL
LIN {X 0,Y 208.679,Z 1223.366,A -85,B 0,C 180,E1 10429.509,E2 10429.509} C_VEL
LIN {X 0,Y 217.47,Z 1224.317,A -85,B 0,C 180,E1 10424.26,E2 10424.26} C_VEL
LIN {X 0,Y 227.641,Z 1223.332,A -85,B 0,C 180,E1 10419.696,E2 10419.696} C_VEL
LIN {X 0,Y 239.357,Z 1220.567,A -85,B 0,C 180,E1 10415.589,E2 10415.589} C_VEL
LIN {X 0,Y 252.595,Z 1215.943,A -85,B 0,C 180,E1 10411.897,E2 10411.897} C_VEL
LIN {X 0,Y 267.085,Z 1209.401,A -85,B 0,C 180,E1 10408.642,E2 10408.642} C_VEL
LIN {X 0,Y 277.267,Z 1203.996,A -85,B 0,C 180,E1 10406.687,E2 10406.687} C_VEL
LIN {X 0,Y 259.167,Z 1215.918,A -85,B 0,C 180,E1 10403.361,E2 10403.361} C_VEL
LIN {X 0,Y 242.314,Z 1226.282,A -85,B 0,C 180,E1 10399.309,E2 10399.309} C_VEL
LIN {X 0,Y 236.895,Z 1229.467,A -85,B 0,C 180,E1 10397.737,E2 10397.737} C_VEL
LIN {X 0,Y 231.704,Z 1232.15,A -85,B 0,C 180,E1 10396.477,E2 10396.477} C_VEL
LIN {X 0,Y 216.46,Z 1238.225,A -85,B 0,C 180,E1 10393.507,E2 10393.507} C_VEL
LIN {X 0,Y 211.739,Z 1240.174,A -85,B 0,C 180,E1 10391.954,E2 10391.954} C_VEL
LIN {X 0,Y 199.632,Z 1245.999,A -85,B 0,C 180,E1 10385.164,E2 10385.164} C_VEL
LIN {X 0,Y 191.587,Z 1249.74,A -85,B 0,C 180,E1 10378.01,E2 10378.01} C_VEL
LIN {X 0,Y 186.967,Z 1251.79,A -85,B 0,C 180,E1 10370.01,E2 10370.01} C_VEL
LIN {X 0,Y 186.061,Z 1252.238,A -85,B 0,C 180,E1 10364.625,E2 10364.625} C_VEL
LIN {X 0,Y 185.576,Z 1261.07,A -85,B 0,C 180,E1 10358.985,E2 10358.985} C_VEL
LIN {X 0,Y 185.765,Z 1267.244,A -85,B 0,C 180,E1 10354.008,E2 10354.008} C_VEL
LIN {X 0,Y 185.793,Z 1271.209,A -85,B 0,C 180,E1 10349.996,E2 10349.996} C_VEL
LIN {X 0,Y 185.302,Z 1274.438,A -85,B 0,C 180,E1 10345.663,E2 10345.663} C_VEL
LIN {X 0,Y 184.874,Z 1277.461,A -85,B 0,C 180,E1 10339.851,E2 10339.851} C_VEL
LIN {X 0,Y 186.435,Z 1279.736,A -85,B 0,C 180,E1 10331.872,E2 10331.872} C_VEL
LIN {X 0,Y 191.462,Z 1280.306,A -85,B 0,C 180,E1 10323.93,E2 10323.93} C_VEL
LIN {X 0,Y 200.829,Z 1279.012,A -85,B 0,C 180,E1 10316.104,E2 10316.104} C_VEL
LIN {X 0,Y 215.19,Z 1275.913,A -85,B 0,C 180,E1 10308.711,E2 10308.711} C_VEL
LIN {X 0,Y 232.043,Z 1271.584,A -85,B 0,C 180,E1 10302.909,E2 10302.909} C_VEL
LIN {X 0,Y 215.182,Z 1273.139,A -85,B 0,C 180,E1 10296.829,E2 10296.829} C_VEL
LIN {X 0,Y 202.135,Z 1272.939,A -85,B 0,C 180,E1 10289.975,E2 10289.975} C_VEL
LIN {X 0,Y 192.967,Z 1271.106,A -85,B 0,C 180,E1 10282.547,E2 10282.547} C_VEL
LIN {X 0,Y 187.599,Z 1267.838,A -85,B 0,C 180,E1 10275.139,E2 10275.139} C_VEL
LIN {X 0,Y 185.14,Z 1263.19,A -85,B 0,C 180,E1 10268.072,E2 10268.072} C_VEL
LIN {X 0,Y 184.422,Z 1257.485,A -85,B 0,C 180,E1 10261.553,E2 10261.553} C_VEL
LIN {X 0,Y 184.353,Z 1251.558,A -85,B 0,C 180,E1 10256.268,E2 10256.268} C_VEL
LIN {X 0,Y 184.725,Z 1243.903,A -85,B 0,C 180,E1 10250.655,E2 10250.655} C_VEL
LIN {X 0,Y 185.875,Z 1234.473,A -85,B 0,C 180,E1 10245.036,E2 10245.036} C_VEL
LIN {X 0,Y 188.248,Z 1222.539,A -85,B 0,C 180,E1 10239.153,E2 10239.153} C_VEL
LIN {X 0,Y 191.754,Z 1209.123,A -85,B 0,C 180,E1 10233.69,E2 10233.69} C_VEL
LIN {X 0,Y 196.242,Z 1194.214,A -85,B 0,C 180,E1 10228.687,E2 10228.687} C_VEL
LIN {X 0,Y 201.892,Z 1176.717,A -85,B 0,C 180,E1 10223.888,E2 10223.888} C_VEL
LIN {X 0,Y 207.801,Z 1158.659,A -85,B 0,C 180,E1 10219.851,E2 10219.851} C_VEL
LIN {X 0,Y 214.073,Z 1139.065,A -85,B 0,C 180,E1 10216.269,E2 10216.269} C_VEL
LIN {X 0,Y 220.512,Z 1117.835,A -85,B 0,C 180,E1 10213.11,E2 10213.11} C_VEL
LIN {X 0,Y 226.841,Z 1095.136,A -85,B 0,C 180,E1 10210.392,E2 10210.392} C_VEL
LIN {X 0,Y 232.686,Z 1071.545,A -85,B 0,C 180,E1 10208.151,E2 10208.151} C_VEL
LIN {X 0,Y 237.93,Z 1046.825,A -85,B 0,C 180,E1 10206.32,E2 10206.32} C_VEL
LIN {X 0,Y 242.412,Z 1021.122,A -85,B 0,C 180,E1 10204.883,E2 10204.883} C_VEL
LIN {X 0,Y 268.137,Z 845.526,A -85,B 0,C 180,E1 10198.028,E2 10198.028} C_VEL
LIN {X 0,Y 257.073,Z 822.429,A -85,B 0,C 180,E1 10194.29,E2 10194.29} C_VEL
LIN {X 0,Y 246.342,Z 801.563,A -85,B 0,C 180,E1 10190.309,E2 10190.309} C_VEL
LIN {X 0,Y 236.562,Z 783.877,A -85,B 0,C 180,E1 10186.328,E2 10186.328} C_VEL
LIN {X 0,Y 227.163,Z 767.891,A -85,B 0,C 180,E1 10182.072,E2 10182.072} C_VEL
LIN {X 0,Y 226.282,Z 767.366,A -85,B 0,C 180,E1 10181.731,E2 10181.731} C_VEL
LIN {X 0,Y 221.064,Z 766.439,A -85,B 0,C 180,E1 10179.835,E2 10179.835} C_VEL
LIN {X 0,Y 223.621,Z 771.983,A -85,B 0,C 180,E1 10175.391,E2 10175.391} C_VEL
LIN {X 0,Y 226.09,Z 777.725,A -85,B 0,C 180,E1 10171.524,E2 10171.524} C_VEL
LIN {X 0,Y 229.39,Z 785.467,A -85,B 0,C 180,E1 10167.005,E2 10167.005} C_VEL
LIN {X 0,Y 233.018,Z 794.705,A -85,B 0,C 180,E1 10162.409,E2 10162.409} C_VEL
LIN {X 0,Y 236.94,Z 805.422,A -85,B 0,C 180,E1 10157.823,E2 10157.823} C_VEL
LIN {X 0,Y 240.925,Z 817.445,A -85,B 0,C 180,E1 10153.363,E2 10153.363} C_VEL
LIN {X 0,Y 244.973,Z 830.992,A -85,B 0,C 180,E1 10148.954,E2 10148.954} C_VEL
LIN {X 0,Y 248.849,Z 845.843,A -85,B 0,C 180,E1 10144.698,E2 10144.698} C_VEL
LIN {X 0,Y 249.486,Z 849.146,A -85,B 0,C 180,E1 10143.845,E2 10143.845} C_VEL
LIN {X 0,Y 235.96,Z 890.935,A -85,B 0,C 180,E1 10137.942,E2 10137.942} C_VEL
LIN {X 0,Y 223.458,Z 933.759,A -85,B 0,C 180,E1 10131.542,E2 10131.542} C_VEL
LIN {X 0,Y 222.822,Z 936.818,A -85,B 0,C 180,E1 10131.137,E2 10131.137} C_VEL
LIN {X 0,Y 222.24,Z 945.424,A -85,B 0,C 180,E1 10130.6,E2 10130.6} C_VEL
LIN {X 0,Y 214.466,Z 1000.305,A -85,B 0,C 180,E1 10127.4,E2 10127.4} C_VEL
LIN {X 0,Y 207.508,Z 1048.089,A -85,B 0,C 180,E1 10123.938,E2 10123.938} C_VEL
LIN {X 0,Y 202.411,Z 1088.094,A -85,B 0,C 180,E1 10120.326,E2 10120.326} C_VEL
LIN {X 0,Y 199.727,Z 1107.126,A -85,B 0,C 180,E1 10118.138,E2 10118.138} C_VEL
LIN {X 0,Y 196.847,Z 1124.661,A -85,B 0,C 180,E1 10115.503,E2 10115.503} C_VEL
LIN {X 0,Y 194.103,Z 1140.116,A -85,B 0,C 180,E1 10112.569,E2 10112.569} C_VEL
LIN {X 0,Y 191.21,Z 1156.17,A -85,B 0,C 180,E1 10108.757,E2 10108.757} C_VEL
LIN {X 0,Y 188.715,Z 1171.086,A -85,B 0,C 180,E1 10104.323,E2 10104.323} C_VEL
LIN {X 0,Y 187.079,Z 1183.579,A -85,B 0,C 180,E1 10099.677,E2 10099.677} C_VEL
LIN {X 0,Y 186.317,Z 1194.062,A -85,B 0,C 180,E1 10094.928,E2 10094.928} C_VEL
LIN {X 0,Y 186.508,Z 1203.562,A -85,B 0,C 180,E1 10089.567,E2 10089.567} C_VEL
LIN {X 0,Y 187.868,Z 1211.094,A -85,B 0,C 180,E1 10084.273,E2 10084.273} C_VEL
LIN {X 0,Y 191.189,Z 1217.744,A -85,B 0,C 180,E1 10078.202,E2 10078.202} C_VEL
LIN {X 0,Y 196.536,Z 1222.274,A -85,B 0,C 180,E1 10072.399,E2 10072.399} C_VEL
LIN {X 0,Y 203.487,Z 1224.811,A -85,B 0,C 180,E1 10067.225,E2 10067.225} C_VEL
LIN {X 0,Y 212.676,Z 1225.673,A -85,B 0,C 180,E1 10062.206,E2 10062.206} C_VEL
LIN {X 0,Y 224.197,Z 1224.605,A -85,B 0,C 180,E1 10057.446,E2 10057.446} C_VEL
LIN {X 0,Y 236.103,Z 1221.959,A -85,B 0,C 180,E1 10053.597,E2 10053.597} C_VEL
LIN {X 0,Y 250.011,Z 1217.433,A -85,B 0,C 180,E1 10050.005,E2 10050.005} C_VEL
LIN {X 0,Y 265.319,Z 1210.954,A -85,B 0,C 180,E1 10046.78,E2 10046.78} C_VEL
LIN {X 0,Y 247.171,Z 1221.552,A -85,B 0,C 180,E1 10043.217,E2 10043.217} C_VEL
LIN {X 0,Y 230.039,Z 1230.893,A -85,B 0,C 180,E1 10038.755,E2 10038.755} C_VEL
LIN {X 0,Y 214.607,Z 1238.737,A -85,B 0,C 180,E1 10033.222,E2 10033.222} C_VEL
LIN {X 0,Y 211.739,Z 1240.174,A -85,B 0,C 180,E1 10031.954,E2 10031.954} C_VEL
LIN {X 0,Y 206.809,Z 1242.119,A -85,B 0,C 180,E1 10030.188,E2 10030.188} C_VEL
LIN {X 0,Y 193.539,Z 1245.559,A -85,B 0,C 180,E1 10026.196,E2 10026.196} C_VEL
LIN {X 0,Y 189.752,Z 1246.644,A -85,B 0,C 180,E1 10024.205,E2 10024.205} C_VEL
LIN {X 0,Y 181.96,Z 1249.6,A -85,B 0,C 180,E1 10016.074,E2 10016.074} C_VEL
LIN {X 0,Y 178.479,Z 1250.502,A -85,B 0,C 180,E1 10007.604,E2 10007.604} C_VEL
LIN {X 0,Y 178.234,Z 1250.548,A -85,B 0,C 180,E1 10004.813,E2 10004.813} C_VEL
LIN {X 0,Y 177.721,Z 1258.854,A -85,B 0,C 180,E1 9999.386,E2 9999.386} C_VEL
LIN {X 0,Y 177.919,Z 1265.739,A -85,B 0,C 180,E1 9993.862,E2 9993.862} C_VEL
LIN {X 0,Y 177.929,Z 1270.074,A -85,B 0,C 180,E1 9989.352,E2 9989.352} C_VEL
LIN {X 0,Y 177.327,Z 1273.514,A -85,B 0,C 180,E1 9984.495,E2 9984.495} C_VEL
LIN {X 0,Y 177.08,Z 1276.57,A -85,B 0,C 180,E1 9978.267,E2 9978.267} C_VEL
LIN {X 0,Y 179.353,Z 1278.943,A -85,B 0,C 180,E1 9969.774,E2 9969.774} C_VEL
LIN {X 0,Y 185.325,Z 1279.539,A -85,B 0,C 180,E1 9961.65,E2 9961.65} C_VEL
LIN {X 0,Y 196.348,Z 1278.381,A -85,B 0,C 180,E1 9953.425,E2 9953.425} C_VEL
LIN {X 0,Y 211.681,Z 1275.627,A -85,B 0,C 180,E1 9946.279,E2 9946.279} C_VEL
LIN {X 0,Y 221.598,Z 1273.425,A -85,B 0,C 180,E1 9942.818,E2 9942.818} C_VEL
LIN {X 0,Y 205.118,Z 1274.012,A -85,B 0,C 180,E1 9936.492,E2 9936.492} C_VEL
LIN {X 0,Y 192.369,Z 1272.95,A -85,B 0,C 180,E1 9929.248,E2 9929.248} C_VEL
LIN {X 0,Y 183.633,Z 1270.277,A -85,B 0,C 180,E1 9921.383,E2 9921.383} C_VEL
LIN {X 0,Y 178.81,Z 1266.18,A -85,B 0,C 180,E1 9913.583,E2 9913.583} C_VEL
LIN {X 0,Y 176.89,Z 1260.991,A -85,B 0,C 180,E1 9906.491,E2 9906.491} C_VEL
LIN {X 0,Y 176.435,Z 1255.249,A -85,B 0,C 180,E1 9900.325,E2 9900.325} C_VEL
LIN {X 0,Y 176.466,Z 1248.333,A -85,B 0,C 180,E1 9894.472,E2 9894.472} C_VEL
LIN {X 0,Y 177.017,Z 1240.38,A -85,B 0,C 180,E1 9888.927,E2 9888.927} C_VEL
LIN {X 0,Y 178.635,Z 1229.616,A -85,B 0,C 180,E1 9882.743,E2 9882.743} C_VEL
LIN {X 0,Y 181.395,Z 1217.474,A -85,B 0,C 180,E1 9876.96,E2 9876.96} C_VEL
LIN {X 0,Y 185.478,Z 1203.087,A -85,B 0,C 180,E1 9871.328,E2 9871.328} C_VEL
LIN {X 0,Y 190.689,Z 1186.745,A -85,B 0,C 180,E1 9866.113,E2 9866.113} C_VEL
LIN {X 0,Y 196.473,Z 1169.42,A -85,B 0,C 180,E1 9861.609,E2 9861.609} C_VEL
LIN {X 0,Y 202.669,Z 1150.896,A -85,B 0,C 180,E1 9857.667,E2 9857.667} C_VEL
LIN {X 0,Y 209.403,Z 1130.042,A -85,B 0,C 180,E1 9854.058,E2 9854.058} C_VEL
LIN {X 0,Y 215.982,Z 1108.127,A -85,B 0,C 180,E1 9851.008,E2 9851.008} C_VEL
LIN {X 0,Y 222.232,Z 1085.27,A -85,B 0,C 180,E1 9848.475,E2 9848.475} C_VEL
LIN {X 0,Y 227.918,Z 1061.494,A -85,B 0,C 180,E1 9846.387,E2 9846.387} C_VEL
LIN {X 0,Y 232.95,Z 1036.705,A -85,B 0,C 180,E1 9844.703,E2 9844.703} C_VEL
LIN {X 0,Y 237.344,Z 1009.931,A -85,B 0,C 180,E1 9843.35,E2 9843.35} C_VEL
LIN {X 0,Y 261.676,Z 848.099,A -85,B 0,C 180,E1 9836.96,E2 9836.96} C_VEL
LIN {X 0,Y 250.581,Z 824.889,A -85,B 0,C 180,E1 9833.054,E2 9833.054} C_VEL
LIN {X 0,Y 240.454,Z 805.025,A -85,B 0,C 180,E1 9829.118,E2 9829.118} C_VEL
LIN {X 0,Y 230.401,Z 786.682,A -85,B 0,C 180,E1 9824.807,E2 9824.807} C_VEL
LIN {X 0,Y 223.519,Z 775.092,A -85,B 0,C 180,E1 9821.57,E2 9821.57} C_VEL
LIN {X 0,Y 216.774,Z 773.827,A -85,B 0,C 180,E1 9819.093,E2 9819.093} C_VEL
LIN {X 0,Y 219.013,Z 779.18,A -85,B 0,C 180,E1 9814.98,E2 9814.98} C_VEL
LIN {X 0,Y 221.606,Z 784.972,A -85,B 0,C 180,E1 9811.038,E2 9811.038} C_VEL
LIN {X 0,Y 224.962,Z 793.552,A -85,B 0,C 180,E1 9806.181,E2 9806.181} C_VEL
LIN {X 0,Y 228.447,Z 802.752,A -85,B 0,C 180,E1 9801.699,E2 9801.699} C_VEL
LIN {X 0,Y 232.061,Z 813.162,A -85,B 0,C 180,E1 9797.31,E2 9797.31} C_VEL
LIN {X 0,Y 235.973,Z 825.607,A -85,B 0,C 180,E1 9792.75,E2 9792.75} C_VEL
LIN {X 0,Y 239.705,Z 838.905,A -85,B 0,C 180,E1 9788.468,E2 9788.468} C_VEL
LIN {X 0,Y 242.795,Z 851.711,A -85,B 0,C 180,E1 9784.798,E2 9784.798} C_VEL
LIN {X 0,Y 228.98,Z 893.068,A -85,B 0,C 180,E1 9778.857,E2 9778.857} C_VEL
LIN {X 0,Y 215.859,Z 936.992,A -85,B 0,C 180,E1 9772.175,E2 9772.175} C_VEL
LIN {X 0,Y 215.207,Z 945.725,A -85,B 0,C 180,E1 9771.603,E2 9771.603} C_VEL
LIN {X 0,Y 207.296,Z 1000.027,A -85,B 0,C 180,E1 9768.361,E2 9768.361} C_VEL
LIN {X 0,Y 200.696,Z 1043.56,A -85,B 0,C 180,E1 9765.13,E2 9765.13} C_VEL
LIN {X 0,Y 194.844,Z 1087.178,A -85,B 0,C 180,E1 9761.061,E2 9761.061} C_VEL
LIN {X 0,Y 192.294,Z 1105.065,A -85,B 0,C 180,E1 9758.99,E2 9758.99} C_VEL
LIN {X 0,Y 189.449,Z 1122.093,A -85,B 0,C 180,E1 9756.425,E2 9756.425} C_VEL
LIN {X 0,Y 186.253,Z 1139.736,A -85,B 0,C 180,E1 9753.018,E2 9753.018} C_VEL
LIN {X 0,Y 183.43,Z 1155.053,A -85,B 0,C 180,E1 9749.298,E2 9749.298} C_VEL
LIN {X 0,Y 181.049,Z 1168.79,A -85,B 0,C 180,E1 9745.167,E2 9745.167} C_VEL
LIN {X 0,Y 179.216,Z 1182.096,A -85,B 0,C 180,E1 9740.238,E2 9740.238} C_VEL
LIN {X 0,Y 178.355,Z 1192.918,A -85,B 0,C 180,E1 9735.277,E2 9735.277} C_VEL
LIN {X 0,Y 178.45,Z 1202.358,A -85,B 0,C 180,E1 9730.003,E2 9730.003} C_VEL
LIN {X 0,Y 179.743,Z 1210.312,A -85,B 0,C 180,E1 9724.467,E2 9724.467} C_VEL
LIN {X 0,Y 182.844,Z 1217.199,A -85,B 0,C 180,E1 9718.433,E2 9718.433} C_VEL
LIN {X 0,Y 188.492,Z 1222.576,A -85,B 0,C 180,E1 9712.072,E2 9712.072} C_VEL
LIN {X 0,Y 196.45,Z 1225.801,A -85,B 0,C 180,E1 9706.159,E2 9706.159} C_VEL
LIN {X 0,Y 206.053,Z 1226.987,A -85,B 0,C 180,E1 9701.027,E2 9701.027} C_VEL
LIN {X 0,Y 217.437,Z 1226.437,A -85,B 0,C 180,E1 9696.417,E2 9696.417} C_VEL
LIN {X 0,Y 231.76,Z 1223.791,A -85,B 0,C 180,E1 9691.949,E2 9691.949} C_VEL
LIN {X 0,Y 247.751,Z 1218.992,A -85,B 0,C 180,E1 9688.082,E2 9688.082} C_VEL
LIN {X 0,Y 253.377,Z 1216.919,A -85,B 0,C 180,E1 9686.88,E2 9686.88} C_VEL
LIN {X 0,Y 235.186,Z 1226.308,A -85,B 0,C 180,E1 9683.055,E2 9683.055} C_VEL
LIN {X 0,Y 217.696,Z 1234.664,A -85,B 0,C 180,E1 9678.073,E2 9678.073} C_VEL
LIN {X 0,Y 203.301,Z 1241.036,A -85,B 0,C 180,E1 9672.355,E2 9672.355} C_VEL
LIN {X 0,Y 190.993,Z 1246.171,A -85,B 0,C 180,E1 9665.155,E2 9665.155} C_VEL
LIN {X 0,Y 189.752,Z 1246.644,A -85,B 0,C 180,E1 9664.205,E2 9664.205} C_VEL
LIN {X 0,Y 185.939,Z 1247.628,A -85,B 0,C 180,E1 9661.966,E2 9661.966} C_VEL
LIN {X 0,Y 175.11,Z 1248.553,A -85,B 0,C 180,E1 9656.586,E2 9656.586} C_VEL
LIN {X 0,Y 172.882,Z 1248.724,A -85,B 0,C 180,E1 9654.33,E2 9654.33} C_VEL
LIN {X 0,Y 170.464,Z 1248.722,A -85,B 0,C 180,E1 9645.649,E2 9645.649} C_VEL
LIN {X 0,Y 170.405,Z 1248.898,A -85,B 0,C 180,E1 9644.957,E2 9644.957} C_VEL
LIN {X 0,Y 169.874,Z 1257.953,A -85,B 0,C 180,E1 9638.798,E2 9638.798} C_VEL
LIN {X 0,Y 170.11,Z 1264.503,A -85,B 0,C 180,E1 9633.365,E2 9633.365} C_VEL
LIN {X 0,Y 170.088,Z 1268.627,A -85,B 0,C 180,E1 9628.985,E2 9628.985} C_VEL
LIN {X 0,Y 169.403,Z 1272.352,A -85,B 0,C 180,E1 9623.556,E2 9623.556} C_VEL
LIN {X 0,Y 169.424,Z 1275.703,A -85,B 0,C 180,E1 9616.341,E2 9616.341} C_VEL
LIN {X 0,Y 172.336,Z 1278.08,A -85,B 0,C 180,E1 9607.84,E2 9607.84} C_VEL
LIN {X 0,Y 179.563,Z 1278.76,A -85,B 0,C 180,E1 9599.179,E2 9599.179} C_VEL
LIN {X 0,Y 192.347,Z 1277.762,A -85,B 0,C 180,E1 9590.635,E2 9590.635} C_VEL
LIN {X 0,Y 208.204,Z 1275.314,A -85,B 0,C 180,E1 9583.911,E2 9583.911} C_VEL
LIN {X 0,Y 211.295,Z 1274.779,A -85,B 0,C 180,E1 9582.771,E2 9582.771} C_VEL
LIN {X 0,Y 195.06,Z 1274.442,A -85,B 0,C 180,E1 9576.122,E2 9576.122} C_VEL
LIN {X 0,Y 182.261,Z 1272.43,A -85,B 0,C 180,E1 9568.151,E2 9568.151} C_VEL
LIN {X 0,Y 174.18,Z 1268.86,A -85,B 0,C 180,E1 9559.797,E2 9559.797} C_VEL
LIN {X 0,Y 170.156,Z 1264.053,A -85,B 0,C 180,E1 9551.869,E2 9551.869} C_VEL
LIN {X 0,Y 168.702,Z 1258.102,A -85,B 0,C 180,E1 9544.419,E2 9544.419} C_VEL
LIN {X 0,Y 168.469,Z 1252.649,A -85,B 0,C 180,E1 9538.98,E2 9538.98} C_VEL
LIN {X 0,Y 168.596,Z 1245.64,A -85,B 0,C 180,E1 9533.188,E2 9533.188} C_VEL
LIN {X 0,Y 169.421,Z 1236.511,A -85,B 0,C 180,E1 9527.04,E2 9527.04} C_VEL
LIN {X 0,Y 171.336,Z 1225.654,A -85,B 0,C 180,E1 9520.925,E2 9520.925} C_VEL
LIN {X 0,Y 174.578,Z 1212.694,A -85,B 0,C 180,E1 9514.923,E2 9514.923} C_VEL
LIN {X 0,Y 179.004,Z 1198.039,A -85,B 0,C 180,E1 9509.348,E2 9509.348} C_VEL
LIN {X 0,Y 184.534,Z 1181.436,A -85,B 0,C 180,E1 9504.183,E2 9504.183} C_VEL
LIN {X 0,Y 190.921,Z 1162.9,A -85,B 0,C 180,E1 9499.502,E2 9499.502} C_VEL
LIN {X 0,Y 197.49,Z 1143.614,A -85,B 0,C 180,E1 9495.556,E2 9495.556} C_VEL
LIN {X 0,Y 204.215,Z 1122.869,A -85,B 0,C 180,E1 9492.132,E2 9492.132} C_VEL
LIN {X 0,Y 210.976,Z 1100.328,A -85,B 0,C 180,E1 9489.151,E2 9489.151} C_VEL
LIN {X 0,Y 217.128,Z 1077.494,A -85,B 0,C 180,E1 9486.747,E2 9486.747} C_VEL
LIN {X 0,Y 222.789,Z 1053.345,A -85,B 0,C 180,E1 9484.753,E2 9484.753} C_VEL
LIN {X 0,Y 227.779,Z 1027.54,A -85,B 0,C 180,E1 9483.139,E2 9483.139} C_VEL
LIN {X 0,Y 237.736,Z 962.61,A -85,B 0,C 180,E1 9480.241,E2 9480.241} C_VEL
LIN {X 0,Y 255.316,Z 850.868,A -85,B 0,C 180,E1 9475.894,E2 9475.894} C_VEL
LIN {X 0,Y 244.468,Z 827.991,A -85,B 0,C 180,E1 9471.886,E2 9471.886} C_VEL
LIN {X 0,Y 234.736,Z 808.745,A -85,B 0,C 180,E1 9467.927,E2 9467.927} C_VEL
LIN {X 0,Y 225.363,Z 791.532,A -85,B 0,C 180,E1 9463.735,E2 9463.735} C_VEL
LIN {X 0,Y 220.174,Z 782.632,A -85,B 0,C 180,E1 9461.204,E2 9461.204} C_VEL
LIN {X 0,Y 214.385,Z 781.787,A -85,B 0,C 180,E1 9459.128,E2 9459.128} C_VEL
LIN {X 0,Y 212.39,Z 781.52,A -85,B 0,C 180,E1 9458.259,E2 9458.259} C_VEL
LIN {X 0,Y 214.147,Z 785.61,A -85,B 0,C 180,E1 9455.093,E2 9455.093} C_VEL
LIN {X 0,Y 216.658,Z 791.538,A -85,B 0,C 180,E1 9451.061,E2 9451.061} C_VEL
LIN {X 0,Y 220.008,Z 800.25,A -85,B 0,C 180,E1 9446.095,E2 9446.095} C_VEL
LIN {X 0,Y 223.617,Z 810.205,A -85,B 0,C 180,E1 9441.259,E2 9441.259} C_VEL
LIN {X 0,Y 227.356,Z 821.625,A -85,B 0,C 180,E1 9436.525,E2 9436.525} C_VEL
LIN {X 0,Y 231.15,Z 834.611,A -85,B 0,C 180,E1 9431.857,E2 9431.857} C_VEL
LIN {X 0,Y 234.596,Z 847.912,A -85,B 0,C 180,E1 9427.653,E2 9427.653} C_VEL
LIN {X 0,Y 235.995,Z 854.7,A -85,B 0,C 180,E1 9425.738,E2 9425.738} C_VEL
LIN {X 0,Y 221.698,Z 896.263,A -85,B 0,C 180,E1 9419.664,E2 9419.664} C_VEL
LIN {X 0,Y 208.868,Z 938.113,A -85,B 0,C 180,E1 9413.188,E2 9413.188} C_VEL
LIN {X 0,Y 208.195,Z 946.229,A -85,B 0,C 180,E1 9412.655,E2 9412.655} C_VEL
LIN {X 0,Y 200.709,Z 996.226,A -85,B 0,C 180,E1 9409.619,E2 9409.619} C_VEL
LIN {X 0,Y 193.255,Z 1043.594,A -85,B 0,C 180,E1 9405.987,E2 9405.987} C_VEL
LIN {X 0,Y 187.447,Z 1085.209,A -85,B 0,C 180,E1 9401.961,E2 9401.961} C_VEL
LIN {X 0,Y 184.677,Z 1104.159,A -85,B 0,C 180,E1 9399.709,E2 9399.709} C_VEL
LIN {X 0,Y 181.407,Z 1123.217,A -85,B 0,C 180,E1 9396.73,E2 9396.73} C_VEL
LIN {X 0,Y 178.14,Z 1140.757,A -85,B 0,C 180,E1 9393.18,E2 9393.18} C_VEL
LIN {X 0,Y 175.218,Z 1156.24,A -85,B 0,C 180,E1 9389.19,E2 9389.19} C_VEL
LIN {X 0,Y 172.774,Z 1170.364,A -85,B 0,C 180,E1 9384.7,E2 9384.7} C_VEL
LIN {X 0,Y 171.1,Z 1182.845,A -85,B 0,C 180,E1 9379.813,E2 9379.813} C_VEL
LIN {X 0,Y 170.316,Z 1194.077,A -85,B 0,C 180,E1 9374.4,E2 9374.4} C_VEL
LIN {X 0,Y 170.626,Z 1203.639,A -85,B 0,C 180,E1 9368.764,E2 9368.764} C_VEL
LIN {X 0,Y 172.537,Z 1212.365,A -85,B 0,C 180,E1 9362.325,E2 9362.325} C_VEL
LIN {X 0,Y 176.382,Z 1219.007,A -85,B 0,C 180,E1 9356.056,E2 9356.056} C_VEL
LIN {X 0,Y 182.526,Z 1223.977,A -85,B 0,C 180,E1 9349.904,E2 9349.904} C_VEL
LIN {X 0,Y 191.602,Z 1227.246,A -85,B 0,C 180,E1 9343.767,E2 9343.767} C_VEL
LIN {X 0,Y 202.315,Z 1228.378,A -85,B 0,C 180,E1 9338.548,E2 9338.548} C_VEL
LIN {X 0,Y 214.782,Z 1227.737,A -85,B 0,C 180,E1 9333.95,E2 9333.95} C_VEL
LIN {X 0,Y 229.059,Z 1225.274,A -85,B 0,C 180,E1 9329.867,E2 9329.867} C_VEL
LIN {X 0,Y 241.423,Z 1221.981,A -85,B 0,C 180,E1 9326.973,E2 9326.973} C_VEL
LIN {X 0,Y 223.24,Z 1230.245,A -85,B 0,C 180,E1 9322.862,E2 9322.862} C_VEL
LIN {X 0,Y 206.048,Z 1237.332,A -85,B 0,C 180,E1 9317.522,E2 9317.522} C_VEL
LIN {X 0,Y 191.597,Z 1242.82,A -85,B 0,C 180,E1 9311.108,E2 9311.108} C_VEL
LIN {X 0,Y 180.188,Z 1246.7,A -85,B 0,C 180,E1 9303.318,E2 9303.318} C_VEL
LIN {X 0,Y 173.387,Z 1248.627,A -85,B 0,C 180,E1 9295.256,E2 9295.256} C_VEL
LIN {X 0,Y 172.882,Z 1248.724,A -85,B 0,C 180,E1 9294.33,E2 9294.33} C_VEL
LIN {X 0,Y 171.094,Z 1248.705,A -85,B 0,C 180,E1 9292.69,E2 9292.69} C_VEL
LIN {X 0,Y 163.707,Z 1247.337,A -85,B 0,C 180,E1 9288.453,E2 9288.453} C_VEL
LIN {X 0,Y 162.767,Z 1246.964,A -85,B 0,C 180,E1 9286.915,E2 9286.915} C_VEL
LIN {X 0,Y 162.652,Z 1246.913,A -85,B 0,C 180,E1 9285.222,E2 9285.222} C_VEL
LIN {X 0,Y 162.045,Z 1256.528,A -85,B 0,C 180,E1 9278.511,E2 9278.511} C_VEL
LIN {X 0,Y 162.317,Z 1262.763,A -85,B 0,C 180,E1 9273.173,E2 9273.173} C_VEL
LIN {X 0,Y 162.319,Z 1266.712,A -85,B 0,C 180,E1 9268.936,E2 9268.936} C_VEL
LIN {X 0,Y 161.635,Z 1270.43,A -85,B 0,C 180,E1 9263.602,E2 9263.602} C_VEL
LIN {X 0,Y 161.739,Z 1274.413,A -85,B 0,C 180,E1 9255.312,E2 9255.312} C_VEL
LIN {X 0,Y 164.905,Z 1276.852,A -85,B 0,C 180,E1 9246.784,E2 9246.784} C_VEL
LIN {X 0,Y 173.395,Z 1277.967,A -85,B 0,C 180,E1 9237.172,E2 9237.172} C_VEL
LIN {X 0,Y 186.151,Z 1277.387,A -85,B 0,C 180,E1 9229.052,E2 9229.052} C_VEL
LIN {X 0,Y 201.065,Z 1275.615,A -85,B 0,C 180,E1 9222.749,E2 9222.749} C_VEL
LIN {X 0,Y 185.021,Z 1274.429,A -85,B 0,C 180,E1 9215.708,E2 9215.708} C_VEL
LIN {X 0,Y 172.606,Z 1271.549,A -85,B 0,C 180,E1 9207.235,E2 9207.235} C_VEL
LIN {X 0,Y 165.063,Z 1267.149,A -85,B 0,C 180,E1 9198.361,E2 9198.361} C_VEL
LIN {X 0,Y 161.646,Z 1261.49,A -85,B 0,C 180,E1 9189.974,E2 9189.974} C_VEL
LIN {X 0,Y 160.653,Z 1255.093,A -85,B 0,C 180,E1 9182.497,E2 9182.497} C_VEL
LIN {X 0,Y 160.539,Z 1248.955,A -85,B 0,C 180,E1 9176.787,E2 9176.787} C_VEL
LIN {X 0,Y 160.848,Z 1241.614,A -85,B 0,C 180,E1 9171.059,E2 9171.059} C_VEL
LIN {X 0,Y 162.172,Z 1231.078,A -85,B 0,C 180,E1 9164.259,E2 9164.259} C_VEL
LIN {X 0,Y 164.733,Z 1219.169,A -85,B 0,C 180,E1 9157.894,E2 9157.894} C_VEL
LIN {X 0,Y 168.748,Z 1205.021,A -85,B 0,C 180,E1 9151.704,E2 9151.704} C_VEL
LIN {X 0,Y 173.902,Z 1189.264,A -85,B 0,C 180,E1 9146.101,E2 9146.101} C_VEL
LIN {X 0,Y 180,Z 1171.842,A -85,B 0,C 180,E1 9141.055,E2 9141.055} C_VEL
LIN {X 0,Y 186.82,Z 1152.516,A -85,B 0,C 180,E1 9136.547,E2 9136.547} C_VEL
LIN {X 0,Y 194.119,Z 1131.101,A -85,B 0,C 180,E1 9132.559,E2 9132.559} C_VEL
LIN {X 0,Y 201.315,Z 1108.464,A -85,B 0,C 180,E1 9129.211,E2 9129.211} C_VEL
LIN {X 0,Y 207.879,Z 1085.749,A -85,B 0,C 180,E1 9126.557,E2 9126.557} C_VEL
LIN {X 0,Y 214.01,Z 1061.429,A -85,B 0,C 180,E1 9124.329,E2 9124.329} C_VEL
LIN {X 0,Y 219.39,Z 1036.182,A -85,B 0,C 180,E1 9122.555,E2 9122.555} C_VEL
LIN {X 0,Y 224.354,Z 1007.177,A -85,B 0,C 180,E1 9121.055,E2 9121.055} C_VEL
LIN {X 0,Y 248.94,Z 853.496,A -85,B 0,C 180,E1 9114.755,E2 9114.755} C_VEL
LIN {X 0,Y 238.205,Z 830.729,A -85,B 0,C 180,E1 9110.617,E2 9110.617} C_VEL
LIN {X 0,Y 228.529,Z 811.443,A -85,B 0,C 180,E1 9106.461,E2 9106.461} C_VEL
LIN {X 0,Y 218.929,Z 793.715,A -85,B 0,C 180,E1 9101.897,E2 9101.897} C_VEL
LIN {X 0,Y 216.859,Z 790.162,A -85,B 0,C 180,E1 9100.856,E2 9100.856} C_VEL
LIN {X 0,Y 212.331,Z 789.557,A -85,B 0,C 180,E1 9099.217,E2 9099.217} C_VEL
LIN {X 0,Y 208.056,Z 788.964,A -85,B 0,C 180,E1 9097.529,E2 9097.529} C_VEL
LIN {X 0,Y 210.53,Z 795.153,A -85,B 0,C 180,E1 9092.998,E2 9092.998} C_VEL
LIN {X 0,Y 213.605,Z 803.019,A -85,B 0,C 180,E1 9088.126,E2 9088.126} C_VEL
LIN {X 0,Y 217.028,Z 812.665,A -85,B 0,C 180,E1 9083.124,E2 9083.124} C_VEL
LIN {X 0,Y 220.433,Z 823.138,A -85,B 0,C 180,E1 9078.491,E2 9078.491} C_VEL
LIN {X 0,Y 223.922,Z 835.017,A -85,B 0,C 180,E1 9073.931,E2 9073.931} C_VEL
LIN {X 0,Y 227.376,Z 848.215,A -85,B 0,C 180,E1 9069.501,E2 9069.501} C_VEL
LIN {X 0,Y 229.318,Z 857.346,A -85,B 0,C 180,E1 9066.763,E2 9066.763} C_VEL
LIN {X 0,Y 214.614,Z 898.888,A -85,B 0,C 180,E1 9060.603,E2 9060.603} C_VEL
LIN {X 0,Y 201.948,Z 939.035,A -85,B 0,C 180,E1 9054.28,E2 9054.28} C_VEL
LIN {X 0,Y 201.165,Z 947.104,A -85,B 0,C 180,E1 9053.74,E2 9053.74} C_VEL
LIN {X 0,Y 193.175,Z 998.548,A -85,B 0,C 180,E1 9050.495,E2 9050.495} C_VEL
LIN {X 0,Y 185.736,Z 1044.398,A -85,B 0,C 180,E1 9046.841,E2 9046.841} C_VEL
LIN {X 0,Y 179.676,Z 1085.96,A -85,B 0,C 180,E1 9042.597,E2 9042.597} C_VEL
LIN {X 0,Y 176.591,Z 1106.15,A -85,B 0,C 180,E1 9040.061,E2 9040.061} C_VEL
LIN {X 0,Y 173.446,Z 1123.854,A -85,B 0,C 180,E1 9037.138,E2 9037.138} C_VEL
LIN {X 0,Y 170.096,Z 1141.25,A -85,B 0,C 180,E1 9033.422,E2 9033.422} C_VEL
LIN {X 0,Y 167.188,Z 1156.391,A -85,B 0,C 180,E1 9029.368,E2 9029.368} C_VEL
LIN {X 0,Y 164.744,Z 1170.324,A -85,B 0,C 180,E1 9024.758,E2 9024.758} C_VEL
LIN {X 0,Y 162.943,Z 1184.049,A -85,B 0,C 180,E1 9019.106,E2 9019.106} C_VEL
LIN {X 0,Y 162.313,Z 1194.994,A -85,B 0,C 180,E1 9013.538,E2 9013.538} C_VEL
LIN {X 0,Y 162.873,Z 1204.864,A -85,B 0,C 180,E1 9007.407,E2 9007.407} C_VEL
LIN {X 0,Y 165.038,Z 1213.097,A -85,B 0,C 180,E1 9001.041,E2 9001.041} C_VEL
LIN {X 0,Y 169.027,Z 1219.544,A -85,B 0,C 180,E1 8994.909,E2 8994.909} C_VEL
LIN {X 0,Y 176.057,Z 1224.962,A -85,B 0,C 180,E1 8988.202,E2 8988.202} C_VEL
LIN {X 0,Y 185.02,Z 1228.195,A -85,B 0,C 180,E1 8982.384,E2 8982.384} C_VEL
LIN {X 0,Y 195.992,Z 1229.698,A -85,B 0,C 180,E1 8977.187,E2 8977.187} C_VEL
LIN {X 0,Y 210.07,Z 1229.359,A -85,B 0,C 180,E1 8972.195,E2 8972.195} C_VEL
LIN {X 0,Y 225.948,Z 1226.965,A -85,B 0,C 180,E1 8967.924,E2 8967.924} C_VEL
LIN {X 0,Y 229.463,Z 1226.2,A -85,B 0,C 180,E1 8967.066,E2 8967.066} C_VEL
LIN {X 0,Y 209.941,Z 1233.873,A -85,B 0,C 180,E1 8962.235,E2 8962.235} C_VEL
LIN {X 0,Y 192.711,Z 1239.866,A -85,B 0,C 180,E1 8956.148,E2 8956.148} C_VEL
LIN {X 0,Y 179.184,Z 1244.074,A -85,B 0,C 180,E1 8949.086,E2 8949.086} C_VEL
LIN {X 0,Y 169.085,Z 1246.629,A -85,B 0,C 180,E1 8940.562,E2 8940.562} C_VEL
LIN {X 0,Y 163.73,Z 1247.336,A -85,B 0,C 180,E1 8931.489,E2 8931.489} C_VEL
LIN {X 0,Y 162.767,Z 1246.964,A -85,B 0,C 180,E1 8926.915,E2 8926.915} C_VEL
LIN {X 0,Y 162.182,Z 1247.572,A -85,B 0,C 180,E1 8925.179,E2 8925.179} C_VEL
LIN {X 0,Y 160.279,Z 1250.165,A -85,B 0,C 180,E1 8922.814,E2 8922.814} C_VEL
LIN {X 0,Y 154.856,Z 1256.656,A -85,B 0,C 180,E1 8917.03,E2 8917.03} C_VEL
LIN {X 0,Y 154.374,Z 1258.722,A -85,B 0,C 180,E1 8915.121,E2 8915.121} C_VEL
LIN {X 0,Y 154.598,Z 1263.855,A -85,B 0,C 180,E1 8909.995,E2 8909.995} C_VEL
LIN {X 0,Y 154.07,Z 1267.51,A -85,B 0,C 180,E1 8905.155,E2 8905.155} C_VEL
LIN {X 0,Y 153.705,Z 1271.738,A -85,B 0,C 180,E1 8897.217,E2 8897.217} C_VEL
LIN {X 0,Y 156.141,Z 1274.951,A -85,B 0,C 180,E1 8888.192,E2 8888.192} C_VEL
LIN {X 0,Y 163.622,Z 1276.822,A -85,B 0,C 180,E1 8878.29,E2 8878.29} C_VEL
LIN {X 0,Y 176.354,Z 1277.093,A -85,B 0,C 180,E1 8869.3,E2 8869.3} C_VEL
LIN {X 0,Y 190.849,Z 1275.986,A -85,B 0,C 180,E1 8862.725,E2 8862.725} C_VEL
LIN {X 0,Y 174.523,Z 1273.872,A -85,B 0,C 180,E1 8854.955,E2 8854.955} C_VEL
LIN {X 0,Y 163.012,Z 1270.237,A -85,B 0,C 180,E1 8846.208,E2 8846.208} C_VEL
LIN {X 0,Y 156.268,Z 1265.156,A -85,B 0,C 180,E1 8837.118,E2 8837.118} C_VEL
LIN {X 0,Y 153.346,Z 1258.772,A -85,B 0,C 180,E1 8828.248,E2 8828.248} C_VEL
LIN {X 0,Y 152.712,Z 1252.729,A -85,B 0,C 180,E1 8821.501,E2 8821.501} C_VEL
LIN {X 0,Y 152.661,Z 1245.728,A -85,B 0,C 180,E1 8815.115,E2 8815.115} C_VEL
LIN {X 0,Y 153.231,Z 1237.144,A -85,B 0,C 180,E1 8808.711,E2 8808.711} C_VEL
LIN {X 0,Y 154.936,Z 1226.376,A -85,B 0,C 180,E1 8801.954,E2 8801.954} C_VEL
LIN {X 0,Y 158.09,Z 1213.54,A -85,B 0,C 180,E1 8795.327,E2 8795.327} C_VEL
LIN {X 0,Y 162.502,Z 1199.221,A -85,B 0,C 180,E1 8789.289,E2 8789.289} C_VEL
LIN {X 0,Y 168.29,Z 1182.54,A -85,B 0,C 180,E1 8783.548,E2 8783.548} C_VEL
LIN {X 0,Y 174.907,Z 1164.276,A -85,B 0,C 180,E1 8778.5,E2 8778.5} C_VEL
LIN {X 0,Y 181.925,Z 1144.761,A -85,B 0,C 180,E1 8774.172,E2 8774.172} C_VEL
LIN {X 0,Y 188.863,Z 1124.665,A -85,B 0,C 180,E1 8770.583,E2 8770.583} C_VEL
LIN {X 0,Y 196.099,Z 1101.901,A -85,B 0,C 180,E1 8767.361,E2 8767.361} C_VEL
LIN {X 0,Y 202.708,Z 1078.817,A -85,B 0,C 180,E1 8764.785,E2 8764.785} C_VEL
LIN {X 0,Y 208.923,Z 1053.735,A -85,B 0,C 180,E1 8762.613,E2 8762.613} C_VEL
LIN {X 0,Y 214.194,Z 1028.115,A -85,B 0,C 180,E1 8760.932,E2 8760.932} C_VEL
LIN {X 0,Y 225.218,Z 960.467,A -85,B 0,C 180,E1 8757.789,E2 8757.789} C_VEL
LIN {X 0,Y 242.624,Z 856.265,A -85,B 0,C 180,E1 8753.601,E2 8753.601} C_VEL
LIN {X 0,Y 232.197,Z 833.896,A -85,B 0,C 180,E1 8749.368,E2 8749.368} C_VEL
LIN {X 0,Y 222.54,Z 814.486,A -85,B 0,C 180,E1 8745.012,E2 8745.012} C_VEL
LIN {X 0,Y 213.484,Z 797.624,A -85,B 0,C 180,E1 8740.467,E2 8740.467} C_VEL
LIN {X 0,Y 203.686,Z 796.61,A -85,B 0,C 180,E1 8736.699,E2 8736.699} C_VEL
LIN {X 0,Y 206.14,Z 802.833,A -85,B 0,C 180,E1 8732.228,E2 8732.228} C_VEL
LIN {X 0,Y 209.108,Z 811.159,A -85,B 0,C 180,E1 8727.263,E2 8727.263} C_VEL
LIN {X 0,Y 212.337,Z 820.664,A -85,B 0,C 180,E1 8722.427,E2 8722.427} C_VEL
LIN {X 0,Y 215.661,Z 831.577,A -85,B 0,C 180,E1 8717.69,E2 8717.69} C_VEL
LIN {X 0,Y 219.049,Z 844.034,A -85,B 0,C 180,E1 8713.018,E2 8713.018} C_VEL
LIN {X 0,Y 222.161,Z 857.121,A -85,B 0,C 180,E1 8708.695,E2 8708.695} C_VEL
LIN {X 0,Y 222.712,Z 859.965,A -85,B 0,C 180,E1 8707.848,E2 8707.848} C_VEL
LIN {X 0,Y 207.285,Z 902.193,A -85,B 0,C 180,E1 8701.479,E2 8701.479} C_VEL
LIN {X 0,Y 195.044,Z 939.727,A -85,B 0,C 180,E1 8695.43,E2 8695.43} C_VEL
LIN {X 0,Y 194.17,Z 947.832,A -85,B 0,C 180,E1 8694.883,E2 8694.883} C_VEL
LIN {X 0,Y 186.101,Z 998.362,A -85,B 0,C 180,E1 8691.622,E2 8691.622} C_VEL
LIN {X 0,Y 178.786,Z 1041.633,A -85,B 0,C 180,E1 8688.059,E2 8688.059} C_VEL
LIN {X 0,Y 172.384,Z 1083.613,A -85,B 0,C 180,E1 8683.65,E2 8683.65} C_VEL
LIN {X 0,Y 169.163,Z 1104.218,A -85,B 0,C 180,E1 8681.003,E2 8681.003} C_VEL
LIN {X 0,Y 166.031,Z 1121.451,A -85,B 0,C 180,E1 8678.118,E2 8678.118} C_VEL
LIN {X 0,Y 162.664,Z 1138.702,A -85,B 0,C 180,E1 8674.439,E2 8674.439} C_VEL
LIN {X 0,Y 159.503,Z 1154.696,A -85,B 0,C 180,E1 8670.1,E2 8670.1} C_VEL
LIN {X 0,Y 156.88,Z 1169.164,A -85,B 0,C 180,E1 8665.184,E2 8665.184} C_VEL
LIN {X 0,Y 155.147,Z 1181.72,A -85,B 0,C 180,E1 8659.973,E2 8659.973} C_VEL
LIN {X 0,Y 154.344,Z 1193.975,A -85,B 0,C 180,E1 8653.678,E2 8653.678} C_VEL
LIN {X 0,Y 154.799,Z 1203.353,A -85,B 0,C 180,E1 8647.796,E2 8647.796} C_VEL
LIN {X 0,Y 157.078,Z 1212.591,A -85,B 0,C 180,E1 8640.729,E2 8640.729} C_VEL
LIN {X 0,Y 161.785,Z 1220.007,A -85,B 0,C 180,E1 8633.613,E2 8633.613} C_VEL
LIN {X 0,Y 168.503,Z 1225.22,A -85,B 0,C 180,E1 8627.317,E2 8627.317} C_VEL
LIN {X 0,Y 178.326,Z 1229.077,A -85,B 0,C 180,E1 8621.022,E2 8621.022} C_VEL
LIN {X 0,Y 191.017,Z 1231.007,A -85,B 0,C 180,E1 8615.243,E2 8615.243} C_VEL
LIN {X 0,Y 205.08,Z 1230.947,A -85,B 0,C 180,E1 8610.499,E2 8610.499} C_VEL
LIN {X 0,Y 217.571,Z 1229.603,A -85,B 0,C 180,E1 8607.16,E2 8607.16} C_VEL
LIN {X 0,Y 198.119,Z 1236.094,A -85,B 0,C 180,E1 8601.928,E2 8601.928} C_VEL
LIN {X 0,Y 181.848,Z 1240.847,A -85,B 0,C 180,E1 8595.62,E2 8595.62} C_VEL
LIN {X 0,Y 168.41,Z 1244.099,A -85,B 0,C 180,E1 8587.694,E2 8587.694} C_VEL
LIN {X 0,Y 159.557,Z 1245.594,A -85,B 0,C 180,E1 8578.845,E2 8578.845} C_VEL
LIN {X 0,Y 155.227,Z 1245.257,A -85,B 0,C 180,E1 8568.755,E2 8568.755} C_VEL
LIN {X 0,Y 154.939,Z 1244.819,A -85,B 0,C 180,E1 8565.529,E2 8565.529} C_VEL
LIN {X 0,Y 154.229,Z 1255.059,A -85,B 0,C 180,E1 8558.195,E2 8558.195} C_VEL
LIN {X 0,Y 154.374,Z 1258.722,A -85,B 0,C 180,E1 8555.121,E2 8555.121} C_VEL
LIN {X 0,Y 153.687,Z 1261.046,A -85,B 0,C 180,E1 8552.822,E2 8552.822} C_VEL
LIN {X 0,Y 150.983,Z 1263.445,A -85,B 0,C 180,E1 8549.515,E2 8549.515} C_VEL
LIN {X 0,Y 146.32,Z 1266.509,A -85,B 0,C 180,E1 8543.49,E2 8543.49} C_VEL
LIN {X 0,Y 146.024,Z 1267.199,A -85,B 0,C 180,E1 8542.178,E2 8542.178} C_VEL
LIN {X 0,Y 146.603,Z 1271.473,A -85,B 0,C 180,E1 8532.941,E2 8532.941} C_VEL
LIN {X 0,Y 151.285,Z 1274.6,A -85,B 0,C 180,E1 8522.863,E2 8522.863} C_VEL
LIN {X 0,Y 161.361,Z 1276.099,A -85,B 0,C 180,E1 8513.048,E2 8513.048} C_VEL
LIN {X 0,Y 177.2,Z 1276.135,A -85,B 0,C 180,E1 8504.218,E2 8504.218} C_VEL
LIN {X 0,Y 180.646,Z 1275.9,A -85,B 0,C 180,E1 8502.692,E2 8502.692} C_VEL
LIN {X 0,Y 164.088,Z 1272.807,A -85,B 0,C 180,E1 8494.098,E2 8494.098} C_VEL
LIN {X 0,Y 153.2,Z 1268.281,A -85,B 0,C 180,E1 8484.69,E2 8484.69} C_VEL
LIN {X 0,Y 147.414,Z 1262.528,A -85,B 0,C 180,E1 8475.339,E2 8475.339} C_VEL
LIN {X 0,Y 145.162,Z 1255.664,A -85,B 0,C 180,E1 8466.327,E2 8466.327} C_VEL
LIN {X 0,Y 144.778,Z 1249.702,A -85,B 0,C 180,E1 8460,E2 8460} C_VEL
LIN {X 0,Y 144.83,Z 1242.537,A -85,B 0,C 180,E1 8453.658,E2 8453.658} C_VEL
LIN {X 0,Y 145.706,Z 1232.824,A -85,B 0,C 180,E1 8446.507,E2 8446.507} C_VEL
LIN {X 0,Y 147.937,Z 1221.215,A -85,B 0,C 180,E1 8439.423,E2 8439.423} C_VEL
LIN {X 0,Y 151.513,Z 1208.192,A -85,B 0,C 180,E1 8432.912,E2 8432.912} C_VEL
LIN {X 0,Y 156.886,Z 1192.065,A -85,B 0,C 180,E1 8426.325,E2 8426.325} C_VEL
LIN {X 0,Y 163.228,Z 1174.697,A -85,B 0,C 180,E1 8420.653,E2 8420.653} C_VEL
LIN {X 0,Y 170.124,Z 1156.238,A -85,B 0,C 180,E1 8415.817,E2 8415.817} C_VEL
LIN {X 0,Y 177.329,Z 1136.517,A -85,B 0,C 180,E1 8411.683,E2 8411.683} C_VEL
LIN {X 0,Y 184.897,Z 1114.462,A -85,B 0,C 180,E1 8408.025,E2 8408.025} C_VEL
LIN {X 0,Y 192.209,Z 1091.088,A -85,B 0,C 180,E1 8404.982,E2 8404.982} C_VEL
LIN {X 0,Y 198.785,Z 1067.307,A -85,B 0,C 180,E1 8402.566,E2 8402.566} C_VEL
LIN {X 0,Y 204.767,Z 1041.66,A -85,B 0,C 180,E1 8400.576,E2 8400.576} C_VEL
LIN {X 0,Y 209.795,Z 1015.35,A -85,B 0,C 180,E1 8399.071,E2 8399.071} C_VEL
LIN {X 0,Y 236.329,Z 858.939,A -85,B 0,C 180,E1 8392.385,E2 8392.385} C_VEL
LIN {X 0,Y 226.185,Z 836.976,A -85,B 0,C 180,E1 8388.062,E2 8388.062} C_VEL
LIN {X 0,Y 216.715,Z 817.747,A -85,B 0,C 180,E1 8383.545,E2 8383.545} C_VEL
LIN {X 0,Y 209.929,Z 805.133,A -85,B 0,C 180,E1 8380.015,E2 8380.015} C_VEL
LIN {X 0,Y 199.309,Z 804.351,A -85,B 0,C 180,E1 8375.835,E2 8375.835} C_VEL
LIN {X 0,Y 202.001,Z 811.585,A -85,B 0,C 180,E1 8370.842,E2 8370.842} C_VEL
LIN {X 0,Y 204.969,Z 820.397,A -85,B 0,C 180,E1 8365.808,E2 8365.808} C_VEL
LIN {X 0,Y 207.933,Z 829.986,A -85,B 0,C 180,E1 8361.152,E2 8361.152} C_VEL
LIN {X 0,Y 211.012,Z 840.88,A -85,B 0,C 180,E1 8356.578,E2 8356.578} C_VEL
LIN {X 0,Y 214.283,Z 854.014,A -85,B 0,C 180,E1 8351.786,E2 8351.786} C_VEL
LIN {X 0,Y 216.122,Z 862.534,A -85,B 0,C 180,E1 8348.993,E2 8348.993} C_VEL
LIN {X 0,Y 200.679,Z 903.581,A -85,B 0,C 180,E1 8342.721,E2 8342.721} C_VEL
LIN {X 0,Y 188.218,Z 940.501,A -85,B 0,C 180,E1 8336.656,E2 8336.656} C_VEL
LIN {X 0,Y 187.181,Z 949.024,A -85,B 0,C 180,E1 8336.081,E2 8336.081} C_VEL
LIN {X 0,Y 179.087,Z 997.887,A -85,B 0,C 180,E1 8332.822,E2 8332.822} C_VEL
LIN {X 0,Y 171.251,Z 1042.759,A -85,B 0,C 180,E1 8328.993,E2 8328.993} C_VEL
LIN {X 0,Y 165.258,Z 1080.392,A -85,B 0,C 180,E1 8324.869,E2 8324.869} C_VEL
LIN {X 0,Y 161.252,Z 1105.086,A -85,B 0,C 180,E1 8321.567,E2 8321.567} C_VEL
LIN {X 0,Y 158.036,Z 1122.262,A -85,B 0,C 180,E1 8318.551,E2 8318.551} C_VEL
LIN {X 0,Y 154.588,Z 1139.328,A -85,B 0,C 180,E1 8314.694,E2 8314.694} C_VEL
LIN {X 0,Y 151.135,Z 1156.458,A -85,B 0,C 180,E1 8309.748,E2 8309.748} C_VEL
LIN {X 0,Y 148.501,Z 1171.217,A -85,B 0,C 180,E1 8304.361,E2 8304.361} C_VEL
LIN {X 0,Y 146.894,Z 1183.834,A -85,B 0,C 180,E1 8298.658,E2 8298.658} C_VEL
LIN {X 0,Y 146.382,Z 1195.527,A -85,B 0,C 180,E1 8292.225,E2 8292.225} C_VEL
LIN {X 0,Y 147.416,Z 1206.059,A -85,B 0,C 180,E1 8285.059,E2 8285.059} C_VEL
LIN {X 0,Y 150.327,Z 1214.468,A -85,B 0,C 180,E1 8278.094,E2 8278.094} C_VEL
LIN {X 0,Y 155.995,Z 1221.758,A -85,B 0,C 180,E1 8270.751,E2 8270.751} C_VEL
LIN {X 0,Y 164.585,Z 1227.236,A -85,B 0,C 180,E1 8263.772,E2 8263.772} C_VEL
LIN {X 0,Y 175.113,Z 1230.672,A -85,B 0,C 180,E1 8257.861,E2 8257.861} C_VEL
LIN {X 0,Y 188.281,Z 1232.446,A -85,B 0,C 180,E1 8252.482,E2 8252.482} C_VEL
LIN {X 0,Y 203.258,Z 1232.366,A -85,B 0,C 180,E1 8247.907,E2 8247.907} C_VEL
LIN {X 0,Y 205.685,Z 1232.24,A -85,B 0,C 180,E1 8247.237,E2 8247.237} C_VEL
LIN {X 0,Y 187.027,Z 1237.433,A -85,B 0,C 180,E1 8241.796,E2 8241.796} C_VEL
LIN {X 0,Y 169.971,Z 1241.409,A -85,B 0,C 180,E1 8234.423,E2 8234.423} C_VEL
LIN {X 0,Y 157.847,Z 1243.494,A -85,B 0,C 180,E1 8226.087,E2 8226.087} C_VEL
LIN {X 0,Y 149.695,Z 1243.939,A -85,B 0,C 180,E1 8215.726,E2 8215.726} C_VEL
LIN {X 0,Y 147.239,Z 1242.703,A -85,B 0,C 180,E1 8205.857,E2 8205.857} C_VEL
LIN {X 0,Y 146.427,Z 1253.545,A -85,B 0,C 180,E1 8197.844,E2 8197.844} C_VEL
LIN {X 0,Y 146.819,Z 1259.9,A -85,B 0,C 180,E1 8191.946,E2 8191.946} C_VEL
LIN {X 0,Y 146.701,Z 1263.615,A -85,B 0,C 180,E1 8187.651,E2 8187.651} C_VEL
LIN {X 0,Y 146.024,Z 1267.199,A -85,B 0,C 180,E1 8182.178,E2 8182.178} C_VEL
LIN {X 0,Y 144.955,Z 1268.508,A -85,B 0,C 180,E1 8179.196,E2 8179.196} C_VEL
LIN {X 0,Y 140.034,Z 1270.459,A -85,B 0,C 180,E1 8170.425,E2 8170.425} C_VEL
LIN {X 0,Y 140.322,Z 1271.094,A -85,B 0,C 180,E1 8168.163,E2 8168.163} C_VEL
LIN {X 0,Y 148.417,Z 1274.138,A -85,B 0,C 180,E1 8156.657,E2 8156.657} C_VEL
LIN {X 0,Y 161.094,Z 1275.334,A -85,B 0,C 180,E1 8147.42,E2 8147.42} C_VEL
LIN {X 0,Y 170.504,Z 1275.367,A -85,B 0,C 180,E1 8142.662,E2 8142.662} C_VEL
LIN {X 0,Y 155.102,Z 1271.748,A -85,B 0,C 180,E1 8134.116,E2 8134.116} C_VEL
LIN {X 0,Y 144.708,Z 1266.655,A -85,B 0,C 180,E1 8124.493,E2 8124.493} C_VEL
LIN {X 0,Y 138.995,Z 1260.039,A -85,B 0,C 180,E1 8114.158,E2 8114.158} C_VEL
LIN {X 0,Y 137.237,Z 1253.586,A -85,B 0,C 180,E1 8105.854,E2 8105.854} C_VEL
LIN {X 0,Y 136.868,Z 1246.863,A -85,B 0,C 180,E1 8098.744,E2 8098.744} C_VEL
LIN {X 0,Y 137.079,Z 1238.555,A -85,B 0,C 180,E1 8091.611,E2 8091.611} C_VEL
LIN {X 0,Y 138.362,Z 1228.105,A -85,B 0,C 180,E1 8084.061,E2 8084.061} C_VEL
LIN {X 0,Y 141.219,Z 1215.524,A -85,B 0,C 180,E1 8076.64,E2 8076.64} C_VEL
LIN {X 0,Y 145.795,Z 1200.708,A -85,B 0,C 180,E1 8069.502,E2 8069.502} C_VEL
LIN {X 0,Y 151.896,Z 1183.731,A -85,B 0,C 180,E1 8062.964,E2 8062.964} C_VEL
LIN {X 0,Y 158.701,Z 1165.926,A -85,B 0,C 180,E1 8057.496,E2 8057.496} C_VEL
LIN {X 0,Y 165.733,Z 1147.54,A -85,B 0,C 180,E1 8052.986,E2 8052.986} C_VEL
LIN {X 0,Y 173.441,Z 1126.535,A -85,B 0,C 180,E1 8048.896,E2 8048.896} C_VEL
LIN {X 0,Y 181.133,Z 1103.87,A -85,B 0,C 180,E1 8045.428,E2 8045.428} C_VEL
LIN {X 0,Y 188.25,Z 1080.543,A -85,B 0,C 180,E1 8042.661,E2 8042.661} C_VEL
LIN {X 0,Y 194.756,Z 1055.953,A -85,B 0,C 180,E1 8040.398,E2 8040.398} C_VEL
LIN {X 0,Y 200.545,Z 1029.767,A -85,B 0,C 180,E1 8038.581,E2 8038.581} C_VEL
LIN {X 0,Y 209.668,Z 977.453,A -85,B 0,C 180,E1 8035.99,E2 8035.99} C_VEL
LIN {X 0,Y 230.079,Z 861.629,A -85,B 0,C 180,E1 8031.113,E2 8031.113} C_VEL
LIN {X 0,Y 219.712,Z 838.967,A -85,B 0,C 180,E1 8026.46,E2 8026.46} C_VEL
LIN {X 0,Y 210.9,Z 821.024,A -85,B 0,C 180,E1 8022.01,E2 8022.01} C_VEL
LIN {X 0,Y 206.478,Z 812.811,A -85,B 0,C 180,E1 8019.621,E2 8019.621} C_VEL
LIN {X 0,Y 194.892,Z 812.054,A -85,B 0,C 180,E1 8015.008,E2 8015.008} C_VEL
LIN {X 0,Y 197.637,Z 820.026,A -85,B 0,C 180,E1 8009.714,E2 8009.714} C_VEL
LIN {X 0,Y 200.584,Z 829.376,A -85,B 0,C 180,E1 8004.569,E2 8004.569} C_VEL
LIN {X 0,Y 203.488,Z 839.537,A -85,B 0,C 180,E1 7999.815,E2 7999.815} C_VEL
LIN {X 0,Y 206.439,Z 851.158,A -85,B 0,C 180,E1 7995.129,E2 7995.129} C_VEL
LIN {X 0,Y 209.188,Z 863.529,A -85,B 0,C 180,E1 7990.747,E2 7990.747} C_VEL
LIN {X 0,Y 209.454,Z 865.556,A -85,B 0,C 180,E1 7990.126,E2 7990.126} C_VEL
LIN {X 0,Y 193.122,Z 907.56,A -85,B 0,C 180,E1 7983.6,E2 7983.6} C_VEL
LIN {X 0,Y 181.406,Z 941.275,A -85,B 0,C 180,E1 7977.934,E2 7977.934} C_VEL
LIN {X 0,Y 179.878,Z 952.074,A -85,B 0,C 180,E1 7977.213,E2 7977.213} C_VEL
LIN {X 0,Y 171.547,Z 1000.716,A -85,B 0,C 180,E1 7973.848,E2 7973.848} C_VEL
LIN {X 0,Y 164.053,Z 1042.088,A -85,B 0,C 180,E1 7970.172,E2 7970.172} C_VEL
LIN {X 0,Y 157.224,Z 1083.097,A -85,B 0,C 180,E1 7965.421,E2 7965.421} C_VEL
LIN {X 0,Y 153.36,Z 1105.913,A -85,B 0,C 180,E1 7962.187,E2 7962.187} C_VEL
LIN {X 0,Y 149.882,Z 1123.688,A -85,B 0,C 180,E1 7958.836,E2 7958.836} C_VEL
LIN {X 0,Y 146.521,Z 1139.847,A -85,B 0,C 180,E1 7954.976,E2 7954.976} C_VEL
LIN {X 0,Y 143.243,Z 1155.727,A -85,B 0,C 180,E1 7950.172,E2 7950.172} C_VEL
LIN {X 0,Y 140.641,Z 1169.917,A -85,B 0,C 180,E1 7944.801,E2 7944.801} C_VEL
LIN {X 0,Y 138.889,Z 1183.527,A -85,B 0,C 180,E1 7938.467,E2 7938.467} C_VEL
LIN {X 0,Y 138.45,Z 1195.286,A -85,B 0,C 180,E1 7931.667,E2 7931.667} C_VEL
LIN {X 0,Y 139.463,Z 1205.127,A -85,B 0,C 180,E1 7924.825,E2 7924.825} C_VEL
LIN {X 0,Y 142.897,Z 1214.667,A -85,B 0,C 180,E1 7916.791,E2 7916.791} C_VEL
LIN {X 0,Y 149.032,Z 1222.11,A -85,B 0,C 180,E1 7909.172,E2 7909.172} C_VEL
LIN {X 0,Y 157.755,Z 1227.676,A -85,B 0,C 180,E1 7902.288,E2 7902.288} C_VEL
LIN {X 0,Y 170.006,Z 1231.758,A -85,B 0,C 180,E1 7895.688,E2 7895.688} C_VEL
LIN {X 0,Y 184.359,Z 1233.764,A -85,B 0,C 180,E1 7890.191,E2 7890.191} C_VEL
LIN {X 0,Y 193.823,Z 1234.082,A -85,B 0,C 180,E1 7887.293,E2 7887.293} C_VEL
LIN {X 0,Y 174.686,Z 1238.42,A -85,B 0,C 180,E1 7881.111,E2 7881.111} C_VEL
LIN {X 0,Y 158.314,Z 1241.203,A -85,B 0,C 180,E1 7873.001,E2 7873.001} C_VEL
LIN {X 0,Y 146.853,Z 1242.268,A -85,B 0,C 180,E1 7863.464,E2 7863.464} C_VEL
LIN {X 0,Y 140.566,Z 1241.495,A -85,B 0,C 180,E1 7852.371,E2 7852.371} C_VEL
LIN {X 0,Y 139.567,Z 1240.51,A -85,B 0,C 180,E1 7846.219,E2 7846.219} C_VEL
LIN {X 0,Y 138.652,Z 1251.363,A -85,B 0,C 180,E1 7837.87,E2 7837.87} C_VEL
LIN {X 0,Y 139.08,Z 1258.012,A -85,B 0,C 180,E1 7831.642,E2 7831.642} C_VEL
LIN {X 0,Y 139.008,Z 1261.443,A -85,B 0,C 180,E1 7827.521,E2 7827.521} C_VEL
LIN {X 0,Y 138.226,Z 1265.902,A -85,B 0,C 180,E1 7820.417,E2 7820.417} C_VEL
LIN {X 0,Y 139.67,Z 1270.491,A -85,B 0,C 180,E1 7809.896,E2 7809.896} C_VEL
LIN {X 0,Y 140.322,Z 1271.094,A -85,B 0,C 180,E1 7808.163,E2 7808.163} C_VEL
LIN {X 0,Y 140.842,Z 1271.885,A -85,B 0,C 180,E1 7805.02,E2 7805.02} C_VEL
LIN {X 0,Y 141.153,Z 1272.582,A -85,B 0,C 180,E1 7796.155,E2 7796.155} C_VEL
LIN {X 0,Y 142.965,Z 1272.958,A -85,B 0,C 180,E1 7793.807,E2 7793.807} C_VEL
LIN {X 0,Y 158.188,Z 1274.353,A -85,B 0,C 180,E1 7783.891,E2 7783.891} C_VEL
LIN {X 0,Y 160.533,Z 1274.421,A -85,B 0,C 180,E1 7782.689,E2 7782.689} C_VEL
LIN {X 0,Y 145.23,Z 1269.965,A -85,B 0,C 180,E1 7773.422,E2 7773.422} C_VEL
LIN {X 0,Y 135.392,Z 1264.025,A -85,B 0,C 180,E1 7763.043,E2 7763.043} C_VEL
LIN {X 0,Y 130.425,Z 1256.579,A -85,B 0,C 180,E1 7751.946,E2 7751.946} C_VEL
LIN {X 0,Y 129.252,Z 1250.098,A -85,B 0,C 180,E1 7743.992,E2 7743.992} C_VEL
LIN {X 0,Y 129.013,Z 1243.604,A -85,B 0,C 180,E1 7737.335,E2 7737.335} C_VEL
LIN {X 0,Y 129.377,Z 1234.79,A -85,B 0,C 180,E1 7729.761,E2 7729.761} C_VEL
LIN {X 0,Y 130.963,Z 1224.196,A -85,B 0,C 180,E1 7722.218,E2 7722.218} C_VEL
LIN {X 0,Y 134.507,Z 1210.365,A -85,B 0,C 180,E1 7714.101,E2 7714.101} C_VEL
LIN {X 0,Y 139.198,Z 1196.335,A -85,B 0,C 180,E1 7707.402,E2 7707.402} C_VEL
LIN {X 0,Y 145.682,Z 1179.183,A -85,B 0,C 180,E1 7700.843,E2 7700.843} C_VEL
LIN {X 0,Y 152.902,Z 1160.841,A -85,B 0,C 180,E1 7695.332,E2 7695.332} C_VEL
LIN {X 0,Y 160.668,Z 1140.89,A -85,B 0,C 180,E1 7690.602,E2 7690.602} C_VEL
LIN {X 0,Y 168.382,Z 1120.038,A -85,B 0,C 180,E1 7686.711,E2 7686.711} C_VEL
LIN {X 0,Y 176.076,Z 1097.382,A -85,B 0,C 180,E1 7683.407,E2 7683.407} C_VEL
LIN {X 0,Y 183.212,Z 1073.787,A -85,B 0,C 180,E1 7680.732,E2 7680.732} C_VEL
LIN {X 0,Y 189.791,Z 1048.543,A -85,B 0,C 180,E1 7678.537,E2 7678.537} C_VEL
LIN {X 0,Y 195.211,Z 1023.129,A -85,B 0,C 180,E1 7676.888,E2 7676.888} C_VEL
LIN {X 0,Y 223.866,Z 864.393,A -85,B 0,C 180,E1 7669.813,E2 7669.813} C_VEL
LIN {X 0,Y 214.232,Z 842.972,A -85,B 0,C 180,E1 7665.224,E2 7665.224} C_VEL
LIN {X 0,Y 205.606,Z 825.117,A -85,B 0,C 180,E1 7660.653,E2 7660.653} C_VEL
LIN {X 0,Y 203.025,Z 820.442,A -85,B 0,C 180,E1 7659.214,E2 7659.214} C_VEL
LIN {X 0,Y 192.757,Z 820.113,A -85,B 0,C 180,E1 7655.146,E2 7655.146} C_VEL
LIN {X 0,Y 190.465,Z 819.933,A -85,B 0,C 180,E1 7654.088,E2 7654.088} C_VEL
LIN {X 0,Y 192.929,Z 827.677,A -85,B 0,C 180,E1 7649.113,E2 7649.113} C_VEL
LIN {X 0,Y 195.648,Z 836.82,A -85,B 0,C 180,E1 7644.137,E2 7644.137} C_VEL
LIN {X 0,Y 198.452,Z 847.388,A -85,B 0,C 180,E1 7639.26,E2 7639.26} C_VEL
LIN {X 0,Y 201.269,Z 859.48,A -85,B 0,C 180,E1 7634.443,E2 7634.443} C_VEL
LIN {X 0,Y 202.996,Z 868.015,A -85,B 0,C 180,E1 7631.406,E2 7631.406} C_VEL
LIN {X 0,Y 186.531,Z 909.145,A -85,B 0,C 180,E1 7624.948,E2 7624.948} C_VEL
LIN {X 0,Y 174.678,Z 942.037,A -85,B 0,C 180,E1 7619.307,E2 7619.307} C_VEL
LIN {X 0,Y 169.83,Z 971.395,A -85,B 0,C 180,E1 7617.364,E2 7617.364} C_VEL
LIN {X 0,Y 161.906,Z 1014.856,A -85,B 0,C 180,E1 7613.972,E2 7613.972} C_VEL
LIN {X 0,Y 154.335,Z 1055.544,A -85,B 0,C 180,E1 7609.862,E2 7609.862} C_VEL
LIN {X 0,Y 148.366,Z 1090.518,A -85,B 0,C 180,E1 7605.331,E2 7605.331} C_VEL
LIN {X 0,Y 144.866,Z 1109.681,A -85,B 0,C 180,E1 7602.296,E2 7602.296} C_VEL
LIN {X 0,Y 141,Z 1128.56,A -85,B 0,C 180,E1 7598.353,E2 7598.353} C_VEL
LIN {X 0,Y 137.553,Z 1144.475,A -85,B 0,C 180,E1 7594.037,E2 7594.037} C_VEL
LIN {X 0,Y 134.316,Z 1160.154,A -85,B 0,C 180,E1 7588.696,E2 7588.696} C_VEL
LIN {X 0,Y 131.926,Z 1174.192,A -85,B 0,C 180,E1 7582.739,E2 7582.739} C_VEL
LIN {X 0,Y 130.627,Z 1187.012,A -85,B 0,C 180,E1 7575.996,E2 7575.996} C_VEL
LIN {X 0,Y 130.676,Z 1197.669,A -85,B 0,C 180,E1 7569.247,E2 7569.247} C_VEL
LIN {X 0,Y 132.566,Z 1208.063,A -85,B 0,C 180,E1 7561.297,E2 7561.297} C_VEL
LIN {X 0,Y 136.957,Z 1216.856,A -85,B 0,C 180,E1 7553.292,E2 7553.292} C_VEL
LIN {X 0,Y 144.321,Z 1224.064,A -85,B 0,C 180,E1 7545.557,E2 7545.557} C_VEL
LIN {X 0,Y 154.271,Z 1229.417,A -85,B 0,C 180,E1 7538.718,E2 7538.718} C_VEL
LIN {X 0,Y 167.13,Z 1233.222,A -85,B 0,C 180,E1 7532.57,E2 7532.57} C_VEL
LIN {X 0,Y 182.058,Z 1235.21,A -85,B 0,C 180,E1 7527.323,E2 7527.323} C_VEL
LIN {X 0,Y 162.474,Z 1238.586,A -85,B 0,C 180,E1 7520.28,E2 7520.28} C_VEL
LIN {X 0,Y 147.374,Z 1240.252,A -85,B 0,C 180,E1 7511.667,E2 7511.667} C_VEL
LIN {X 0,Y 136.688,Z 1240.249,A -85,B 0,C 180,E1 7500.794,E2 7500.794} C_VEL
LIN {X 0,Y 132.255,Z 1238.523,A -85,B 0,C 180,E1 7489.423,E2 7489.423} C_VEL
LIN {X 0,Y 132.018,Z 1237.964,A -85,B 0,C 180,E1 7486.72,E2 7486.72} C_VEL
LIN {X 0,Y 130.85,Z 1247.108,A -85,B 0,C 180,E1 7479.672,E2 7479.672} C_VEL
LIN {X 0,Y 131.282,Z 1254.695,A -85,B 0,C 180,E1 7472.613,E2 7472.613} C_VEL
LIN {X 0,Y 131.43,Z 1258.531,A -85,B 0,C 180,E1 7468.25,E2 7468.25} C_VEL
LIN {X 0,Y 130.665,Z 1262.833,A -85,B 0,C 180,E1 7461.634,E2 7461.634} C_VEL
LIN {X 0,Y 131.348,Z 1267.476,A -85,B 0,C 180,E1 7451.807,E2 7451.807} C_VEL
LIN {X 0,Y 136.937,Z 1271.41,A -85,B 0,C 180,E1 7440.224,E2 7440.224} C_VEL
LIN {X 0,Y 142.965,Z 1272.958,A -85,B 0,C 180,E1 7433.807,E2 7433.807} C_VEL
LIN {X 0,Y 144.287,Z 1273.156,A -85,B 0,C 180,E1 7431.785,E2 7431.785} C_VEL
LIN {X 0,Y 145.527,Z 1272.71,A -85,B 0,C 180,E1 7426.085,E2 7426.085} C_VEL
LIN {X 0,Y 147.372,Z 1272.785,A -85,B 0,C 180,E1 7424.485,E2 7424.485} C_VEL
LIN {X 0,Y 150.508,Z 1273.023,A -85,B 0,C 180,E1 7422.659,E2 7422.659} C_VEL
LIN {X 0,Y 135.742,Z 1267.823,A -85,B 0,C 180,E1 7412.879,E2 7412.879} C_VEL
LIN {X 0,Y 126.203,Z 1260.95,A -85,B 0,C 180,E1 7401.374,E2 7401.374} C_VEL
LIN {X 0,Y 122.299,Z 1253.748,A -85,B 0,C 180,E1 7390.839,E2 7390.839} C_VEL
LIN {X 0,Y 121.345,Z 1246.685,A -85,B 0,C 180,E1 7382.361,E2 7382.361} C_VEL
LIN {X 0,Y 121.192,Z 1239.589,A -85,B 0,C 180,E1 7375.267,E2 7375.267} C_VEL
LIN {X 0,Y 121.794,Z 1230.624,A -85,B 0,C 180,E1 7367.675,E2 7367.675} C_VEL
LIN {X 0,Y 124.041,Z 1218.602,A -85,B 0,C 180,E1 7359.226,E2 7359.226} C_VEL
LIN {X 0,Y 127.927,Z 1205.292,A -85,B 0,C 180,E1 7351.524,E2 7351.524} C_VEL
LIN {X 0,Y 133.565,Z 1189.656,A -85,B 0,C 180,E1 7344.273,E2 7344.273} C_VEL
LIN {X 0,Y 140.396,Z 1172.454,A -85,B 0,C 180,E1 7337.974,E2 7337.974} C_VEL
LIN {X 0,Y 148.006,Z 1153.745,A -85,B 0,C 180,E1 7332.576,E2 7332.576} C_VEL
LIN {X 0,Y 156.17,Z 1133.119,A -85,B 0,C 180,E1 7327.932,E2 7327.932} C_VEL
LIN {X 0,Y 164.489,Z 1110.607,A -85,B 0,C 180,E1 7324.009,E2 7324.009} C_VEL
LIN {X 0,Y 172.365,Z 1087.061,A -85,B 0,C 180,E1 7320.846,E2 7320.846} C_VEL
LIN {X 0,Y 179.493,Z 1062.658,A -85,B 0,C 180,E1 7318.338,E2 7318.338} C_VEL
LIN {X 0,Y 185.877,Z 1036.611,A -85,B 0,C 180,E1 7316.321,E2 7316.321} C_VEL
LIN {X 0,Y 191.787,Z 1006.672,A -85,B 0,C 180,E1 7314.636,E2 7314.636} C_VEL
LIN {X 0,Y 217.717,Z 867.087,A -85,B 0,C 180,E1 7308.444,E2 7308.444} C_VEL
LIN {X 0,Y 208.35,Z 846.06,A -85,B 0,C 180,E1 7303.746,E2 7303.746} C_VEL
LIN {X 0,Y 200.367,Z 829.274,A -85,B 0,C 180,E1 7299.232,E2 7299.232} C_VEL
LIN {X 0,Y 199.569,Z 828.032,A -85,B 0,C 180,E1 7298.794,E2 7298.794} C_VEL
LIN {X 0,Y 188.524,Z 827.918,A -85,B 0,C 180,E1 7294.353,E2 7294.353} C_VEL
LIN {X 0,Y 185.98,Z 827.903,A -85,B 0,C 180,E1 7293.171,E2 7293.171} C_VEL
LIN {X 0,Y 188.211,Z 835.352,A -85,B 0,C 180,E1 7288.482,E2 7288.482} C_VEL
LIN {X 0,Y 190.834,Z 844.96,A -85,B 0,C 180,E1 7283.385,E2 7283.385} C_VEL
LIN {X 0,Y 193.509,Z 856.063,A -85,B 0,C 180,E1 7278.378,E2 7278.378} C_VEL
LIN {X 0,Y 195.996,Z 867.981,A -85,B 0,C 180,E1 7273.709,E2 7273.709} C_VEL
LIN {X 0,Y 196.502,Z 870.783,A -85,B 0,C 180,E1 7272.713,E2 7272.713} C_VEL
LIN {X 0,Y 179.356,Z 912.203,A -85,B 0,C 180,E1 7266.105,E2 7266.105} C_VEL
LIN {X 0,Y 167.981,Z 942.863,A -85,B 0,C 180,E1 7260.747,E2 7260.747} C_VEL
LIN {X 0,Y 159.004,Z 993.217,A -85,B 0,C 180,E1 7257.192,E2 7257.192} C_VEL
LIN {X 0,Y 150.658,Z 1036.218,A -85,B 0,C 180,E1 7253.264,E2 7253.264} C_VEL
LIN {X 0,Y 143.965,Z 1072.321,A -85,B 0,C 180,E1 7248.901,E2 7248.901} C_VEL
LIN {X 0,Y 138.354,Z 1103.385,A -85,B 0,C 180,E1 7244.249,E2 7244.249} C_VEL
LIN {X 0,Y 134.748,Z 1120.911,A -85,B 0,C 180,E1 7240.768,E2 7240.768} C_VEL
LIN {X 0,Y 130.919,Z 1138.265,A -85,B 0,C 180,E1 7236.293,E2 7236.293} C_VEL
LIN {X 0,Y 127.33,Z 1154.814,A -85,B 0,C 180,E1 7230.846,E2 7230.846} C_VEL
LIN {X 0,Y 124.394,Z 1170.546,A -85,B 0,C 180,E1 7224.201,E2 7224.201} C_VEL
LIN {X 0,Y 122.801,Z 1184.132,A -85,B 0,C 180,E1 7217.045,E2 7217.045} C_VEL
LIN {X 0,Y 122.726,Z 1195.981,A -85,B 0,C 180,E1 7209.378,E2 7209.378} C_VEL
LIN {X 0,Y 124.478,Z 1206.302,A -85,B 0,C 180,E1 7201.381,E2 7201.381} C_VEL
LIN {X 0,Y 128.905,Z 1215.64,A -85,B 0,C 180,E1 7192.871,E2 7192.871} C_VEL
LIN {X 0,Y 136.45,Z 1223.402,A -85,B 0,C 180,E1 7184.704,E2 7184.704} C_VEL
LIN {X 0,Y 147.763,Z 1229.723,A -85,B 0,C 180,E1 7176.953,E2 7176.953} C_VEL
LIN {X 0,Y 160.597,Z 1233.761,A -85,B 0,C 180,E1 7170.946,E2 7170.946} C_VEL
LIN {X 0,Y 170.417,Z 1235.643,A -85,B 0,C 180,E1 7167.338,E2 7167.338} C_VEL
LIN {X 0,Y 151.645,Z 1237.898,A -85,B 0,C 180,E1 7159.886,E2 7159.886} C_VEL
LIN {X 0,Y 136.22,Z 1238.643,A -85,B 0,C 180,E1 7149.679,E2 7149.679} C_VEL
LIN {X 0,Y 127.455,Z 1237.673,A -85,B 0,C 180,E1 7138.52,E2 7138.52} C_VEL
LIN {X 0,Y 124.497,Z 1235.387,A -85,B 0,C 180,E1 7127.28,E2 7127.28} C_VEL
LIN {X 0,Y 123.135,Z 1242.99,A -85,B 0,C 180,E1 7121.231,E2 7121.231} C_VEL
LIN {X 0,Y 123.443,Z 1251.21,A -85,B 0,C 180,E1 7113.709,E2 7113.709} C_VEL
LIN {X 0,Y 123.81,Z 1255.753,A -85,B 0,C 180,E1 7108.605,E2 7108.605} C_VEL
LIN {X 0,Y 123.198,Z 1259.493,A -85,B 0,C 180,E1 7103.001,E2 7103.001} C_VEL
LIN {X 0,Y 123.402,Z 1264.53,A -85,B 0,C 180,E1 7092.964,E2 7092.964} C_VEL
LIN {X 0,Y 128.827,Z 1269.113,A -85,B 0,C 180,E1 7080.209,E2 7080.209} C_VEL
LIN {X 0,Y 140.234,Z 1272.006,A -85,B 0,C 180,E1 7069,E2 7069} C_VEL
LIN {X 0,Y 147.372,Z 1272.785,A -85,B 0,C 180,E1 7064.485,E2 7064.485} C_VEL
LIN {X 0,Y 147.735,Z 1272.708,A -85,B 0,C 180,E1 7063.585,E2 7063.585} C_VEL
LIN {X 0,Y 146.416,Z 1272.285,A -85,B 0,C 180,E1 7062.441,E2 7062.441} C_VEL
LIN {X 0,Y 142.925,Z 1271.373,A -85,B 0,C 180,E1 7061.048,E2 7061.048} C_VEL
LIN {X 0,Y 134.239,Z 1268.907,A -85,B 0,C 180,E1 7058.354,E2 7058.354} C_VEL
LIN {X 0,Y 132.049,Z 1268.137,A -85,B 0,C 180,E1 7057.137,E2 7057.137} C_VEL
LIN {X 0,Y 120.64,Z 1261.275,A -85,B 0,C 180,E1 7045.53,E2 7045.53} C_VEL
LIN {X 0,Y 115.11,Z 1253.462,A -85,B 0,C 180,E1 7033.564,E2 7033.564} C_VEL
LIN {X 0,Y 113.698,Z 1246.454,A -85,B 0,C 180,E1 7024.54,E2 7024.54} C_VEL
LIN {X 0,Y 113.377,Z 1239.947,A -85,B 0,C 180,E1 7017.473,E2 7017.473} C_VEL
LIN {X 0,Y 113.664,Z 1231.716,A -85,B 0,C 180,E1 7009.867,E2 7009.867} C_VEL
LIN {X 0,Y 115.632,Z 1219.544,A -85,B 0,C 180,E1 7000.501,E2 7000.501} C_VEL
LIN {X 0,Y 119.449,Z 1206.091,A -85,B 0,C 180,E1 6992.046,E2 6992.046} C_VEL
LIN {X 0,Y 125.085,Z 1190.594,A -85,B 0,C 180,E1 6984.3,E2 6984.3} C_VEL
LIN {X 0,Y 132.163,Z 1173.206,A -85,B 0,C 180,E1 6977.479,E2 6977.479} C_VEL
LIN {X 0,Y 140.046,Z 1154.432,A -85,B 0,C 180,E1 6971.746,E2 6971.746} C_VEL
LIN {X 0,Y 148.726,Z 1133.19,A -85,B 0,C 180,E1 6966.758,E2 6966.758} C_VEL
LIN {X 0,Y 157.318,Z 1110.69,A -85,B 0,C 180,E1 6962.706,E2 6962.706} C_VEL
LIN {X 0,Y 165.4,Z 1087.205,A -85,B 0,C 180,E1 6959.48,E2 6959.48} C_VEL
LIN {X 0,Y 172.902,Z 1062.208,A -85,B 0,C 180,E1 6956.87,E2 6956.87} C_VEL
LIN {X 0,Y 179.352,Z 1036.625,A -85,B 0,C 180,E1 6954.86,E2 6954.86} C_VEL
LIN {X 0,Y 185.409,Z 1006.888,A -85,B 0,C 180,E1 6953.16,E2 6953.16} C_VEL
LIN {X 0,Y 211.602,Z 869.765,A -85,B 0,C 180,E1 6947.004,E2 6947.004} C_VEL
LIN {X 0,Y 202.848,Z 849.816,A -85,B 0,C 180,E1 6942.349,E2 6942.349} C_VEL
LIN {X 0,Y 196.182,Z 835.66,A -85,B 0,C 180,E1 6938.423,E2 6938.423} C_VEL
LIN {X 0,Y 184.554,Z 835.795,A -85,B 0,C 180,E1 6933.636,E2 6933.636} C_VEL
LIN {X 0,Y 181.493,Z 835.97,A -85,B 0,C 180,E1 6932.254,E2 6932.254} C_VEL
LIN {X 0,Y 183.731,Z 844.264,A -85,B 0,C 180,E1 6927.197,E2 6927.197} C_VEL
LIN {X 0,Y 186.097,Z 853.885,A -85,B 0,C 180,E1 6922.285,E2 6922.285} C_VEL
LIN {X 0,Y 188.448,Z 864.917,A -85,B 0,C 180,E1 6917.44,E2 6917.44} C_VEL
LIN {X 0,Y 189.968,Z 873.69,A -85,B 0,C 180,E1 6914.069,E2 6914.069} C_VEL
LIN {X 0,Y 171.907,Z 916.137,A -85,B 0,C 180,E1 6907.207,E2 6907.207} C_VEL
LIN {X 0,Y 161.375,Z 943.715,A -85,B 0,C 180,E1 6902.291,E2 6902.291} C_VEL
LIN {X 0,Y 151.527,Z 996.581,A -85,B 0,C 180,E1 6898.46,E2 6898.46} C_VEL
LIN {X 0,Y 143.299,Z 1037.136,A -85,B 0,C 180,E1 6894.552,E2 6894.552} C_VEL
LIN {X 0,Y 135.995,Z 1075.146,A -85,B 0,C 180,E1 6889.692,E2 6889.692} C_VEL
LIN {X 0,Y 130.56,Z 1103.736,A -85,B 0,C 180,E1 6885.106,E2 6885.106} C_VEL
LIN {X 0,Y 126.653,Z 1121.979,A -85,B 0,C 180,E1 6881.24,E2 6881.24} C_VEL
LIN {X 0,Y 122.728,Z 1139.233,A -85,B 0,C 180,E1 6876.495,E2 6876.495} C_VEL
LIN {X 0,Y 119.032,Z 1155.87,A -85,B 0,C 180,E1 6870.545,E2 6870.545} C_VEL
LIN {X 0,Y 116.133,Z 1171.736,A -85,B 0,C 180,E1 6863.332,E2 6863.332} C_VEL
LIN {X 0,Y 114.758,Z 1185.089,A -85,B 0,C 180,E1 6855.671,E2 6855.671} C_VEL
LIN {X 0,Y 115.016,Z 1196.901,A -85,B 0,C 180,E1 6847.493,E2 6847.493} C_VEL
LIN {X 0,Y 117.721,Z 1208.235,A -85,B 0,C 180,E1 6838.053,E2 6838.053} C_VEL
LIN {X 0,Y 123.243,Z 1217.318,A -85,B 0,C 180,E1 6829.245,E2 6829.245} C_VEL
LIN {X 0,Y 132.017,Z 1224.95,A -85,B 0,C 180,E1 6820.993,E2 6820.993} C_VEL
LIN {X 0,Y 144.722,Z 1231.232,A -85,B 0,C 180,E1 6813.315,E2 6813.315} C_VEL
LIN {X 0,Y 159.069,Z 1235.313,A -85,B 0,C 180,E1 6807.374,E2 6807.374} C_VEL
LIN {X 0,Y 140.336,Z 1236.673,A -85,B 0,C 180,E1 6799.037,E2 6799.037} C_VEL
LIN {X 0,Y 126.213,Z 1236.386,A -85,B 0,C 180,E1 6788.157,E2 6788.157} C_VEL
LIN {X 0,Y 118.435,Z 1234.45,A -85,B 0,C 180,E1 6775.398,E2 6775.398} C_VEL
LIN {X 0,Y 117.01,Z 1232.753,A -85,B 0,C 180,E1 6767.909,E2 6767.909} C_VEL
LIN {X 0,Y 115.399,Z 1240.455,A -85,B 0,C 180,E1 6761.488,E2 6761.488} C_VEL
LIN {X 0,Y 115.764,Z 1248.863,A -85,B 0,C 180,E1 6753.459,E2 6753.459} C_VEL
LIN {X 0,Y 116.2,Z 1253.189,A -85,B 0,C 180,E1 6748.514,E2 6748.514} C_VEL
LIN {X 0,Y 115.596,Z 1257.109,A -85,B 0,C 180,E1 6742.538,E2 6742.538} C_VEL
LIN {X 0,Y 116.103,Z 1262.51,A -85,B 0,C 180,E1 6731.323,E2 6731.323} C_VEL
LIN {X 0,Y 122.022,Z 1267.249,A -85,B 0,C 180,E1 6718.363,E2 6718.363} C_VEL
LIN {X 0,Y 134.864,Z 1270.446,A -85,B 0,C 180,E1 6706.402,E2 6706.402} C_VEL
LIN {X 0,Y 140.725,Z 1271.255,A -85,B 0,C 180,E1 6702.712,E2 6702.712} C_VEL
LIN {X 0,Y 132.049,Z 1268.137,A -85,B 0,C 180,E1 6697.137,E2 6697.137} C_VEL
LIN {X 0,Y 127.603,Z 1266.348,A -85,B 0,C 180,E1 6694.44,E2 6694.44} C_VEL
LIN {X 0,Y 114.289,Z 1260.055,A -85,B 0,C 180,E1 6687.168,E2 6687.168} C_VEL
LIN {X 0,Y 111.628,Z 1257.959,A -85,B 0,C 180,E1 6684.248,E2 6684.248} C_VEL
LIN {X 0,Y 107.023,Z 1250.164,A -85,B 0,C 180,E1 6672.409,E2 6672.409} C_VEL
LIN {X 0,Y 105.81,Z 1242.648,A -85,B 0,C 180,E1 6662.708,E2 6662.708} C_VEL
LIN {X 0,Y 105.589,Z 1234.97,A -85,B 0,C 180,E1 6654.566,E2 6654.566} C_VEL
LIN {X 0,Y 106.399,Z 1225.264,A -85,B 0,C 180,E1 6645.857,E2 6645.857} C_VEL
LIN {X 0,Y 109.285,Z 1212.295,A -85,B 0,C 180,E1 6636.213,E2 6636.213} C_VEL
LIN {X 0,Y 114.052,Z 1198.076,A -85,B 0,C 180,E1 6627.671,E2 6627.671} C_VEL
LIN {X 0,Y 121.03,Z 1180.713,A -85,B 0,C 180,E1 6619.569,E2 6619.569} C_VEL
LIN {X 0,Y 128.508,Z 1163.338,A -85,B 0,C 180,E1 6613.322,E2 6613.322} C_VEL
LIN {X 0,Y 137.086,Z 1143.395,A -85,B 0,C 180,E1 6607.79,E2 6607.79} C_VEL
LIN {X 0,Y 145.866,Z 1121.975,A -85,B 0,C 180,E1 6603.249,E2 6603.249} C_VEL
LIN {X 0,Y 154.544,Z 1098.771,A -85,B 0,C 180,E1 6599.516,E2 6599.516} C_VEL
LIN {X 0,Y 162.635,Z 1074.421,A -85,B 0,C 180,E1 6596.55,E2 6596.55} C_VEL
LIN {X 0,Y 169.726,Z 1049.556,A -85,B 0,C 180,E1 6594.263,E2 6594.263} C_VEL
LIN {X 0,Y 175.724,Z 1023.877,A -85,B 0,C 180,E1 6592.518,E2 6592.518} C_VEL
LIN {X 0,Y 205.602,Z 872.661,A -85,B 0,C 180,E1 6585.55,E2 6585.55} C_VEL
LIN {X 0,Y 197.326,Z 853.359,A -85,B 0,C 180,E1 6580.851,E2 6580.851} C_VEL
LIN {X 0,Y 192.796,Z 843.455,A -85,B 0,C 180,E1 6578.053,E2 6578.053} C_VEL
LIN {X 0,Y 183.164,Z 843.617,A -85,B 0,C 180,E1 6574.074,E2 6574.074} C_VEL
LIN {X 0,Y 176.905,Z 844.202,A -85,B 0,C 180,E1 6571.227,E2 6571.227} C_VEL
LIN {X 0,Y 179.024,Z 852.829,A -85,B 0,C 180,E1 6566.161,E2 6566.161} C_VEL
LIN {X 0,Y 181.258,Z 863.041,A -85,B 0,C 180,E1 6561.119,E2 6561.119} C_VEL
LIN {X 0,Y 183.443,Z 874.777,A -85,B 0,C 180,E1 6556.128,E2 6556.128} C_VEL
LIN {X 0,Y 183.681,Z 876.173,A -85,B 0,C 180,E1 6555.584,E2 6555.584} C_VEL
LIN {X 0,Y 165.979,Z 916.374,A -85,B 0,C 180,E1 6549.028,E2 6549.028} C_VEL
LIN {X 0,Y 154.835,Z 944.401,A -85,B 0,C 180,E1 6543.944,E2 6543.944} C_VEL
LIN {X 0,Y 145.083,Z 994.775,A -85,B 0,C 180,E1 6540.246,E2 6540.246} C_VEL
LIN {X 0,Y 136.277,Z 1036.75,A -85,B 0,C 180,E1 6536.116,E2 6536.116} C_VEL
LIN {X 0,Y 129.282,Z 1071.379,A -85,B 0,C 180,E1 6531.547,E2 6531.547} C_VEL
LIN {X 0,Y 122.831,Z 1103.785,A -85,B 0,C 180,E1 6526.09,E2 6526.09} C_VEL
LIN {X 0,Y 118.985,Z 1121.202,A -85,B 0,C 180,E1 6522.243,E2 6522.243} C_VEL
LIN {X 0,Y 114.731,Z 1139.213,A -85,B 0,C 180,E1 6516.966,E2 6516.966} C_VEL
LIN {X 0,Y 110.808,Z 1156.554,A -85,B 0,C 180,E1 6510.353,E2 6510.353} C_VEL
LIN {X 0,Y 108.159,Z 1170.999,A -85,B 0,C 180,E1 6503.271,E2 6503.271} C_VEL
LIN {X 0,Y 106.824,Z 1184.402,A -85,B 0,C 180,E1 6495.194,E2 6495.194} C_VEL
LIN {X 0,Y 107.257,Z 1196.328,A -85,B 0,C 180,E1 6486.423,E2 6486.423} C_VEL
LIN {X 0,Y 109.891,Z 1206.798,A -85,B 0,C 180,E1 6477.392,E2 6477.392} C_VEL
LIN {X 0,Y 116.065,Z 1216.821,A -85,B 0,C 180,E1 6467.563,E2 6467.563} C_VEL
LIN {X 0,Y 125.958,Z 1225.097,A -85,B 0,C 180,E1 6458.582,E2 6458.582} C_VEL
LIN {X 0,Y 138.794,Z 1231.426,A -85,B 0,C 180,E1 6451.139,E2 6451.139} C_VEL
LIN {X 0,Y 147.626,Z 1234.388,A -85,B 0,C 180,E1 6447.294,E2 6447.294} C_VEL
LIN {X 0,Y 129.199,Z 1234.761,A -85,B 0,C 180,E1 6437.974,E2 6437.974} C_VEL
LIN {X 0,Y 116.102,Z 1233.546,A -85,B 0,C 180,E1 6425.838,E2 6425.838} C_VEL
LIN {X 0,Y 110.088,Z 1230.667,A -85,B 0,C 180,E1 6412.114,E2 6412.114} C_VEL
LIN {X 0,Y 109.624,Z 1229.878,A -85,B 0,C 180,E1 6408.609,E2 6408.609} C_VEL
LIN {X 0,Y 107.729,Z 1237.151,A -85,B 0,C 180,E1 6402.318,E2 6402.318} C_VEL
LIN {X 0,Y 108.095,Z 1246.469,A -85,B 0,C 180,E1 6393.174,E2 6393.174} C_VEL
LIN {X 0,Y 108.611,Z 1250.946,A -85,B 0,C 180,E1 6387.883,E2 6387.883} C_VEL
LIN {X 0,Y 108.019,Z 1254.85,A -85,B 0,C 180,E1 6381.476,E2 6381.476} C_VEL
LIN {X 0,Y 109.178,Z 1260.819,A -85,B 0,C 180,E1 6368.503,E2 6368.503} C_VEL
LIN {X 0,Y 116.164,Z 1265.435,A -85,B 0,C 180,E1 6355.375,E2 6355.375} C_VEL
LIN {X 0,Y 131.032,Z 1269.024,A -85,B 0,C 180,E1 6342.778,E2 6342.778} C_VEL
LIN {X 0,Y 116.937,Z 1262.32,A -85,B 0,C 180,E1 6331.439,E2 6331.439} C_VEL
LIN {X 0,Y 111.628,Z 1257.959,A -85,B 0,C 180,E1 6324.248,E2 6324.248} C_VEL
LIN {X 0,Y 108.826,Z 1255.471,A -85,B 0,C 180,E1 6320.74,E2 6320.74} C_VEL
LIN {X 0,Y 101.773,Z 1249.318,A -85,B 0,C 180,E1 6313.888,E2 6313.888} C_VEL
LIN {X 0,Y 98.765,Z 1245.037,A -85,B 0,C 180,E1 6308.92,E2 6308.92} C_VEL
LIN {X 0,Y 98.516,Z 1244.153,A -85,B 0,C 180,E1 6307.728,E2 6307.728} C_VEL
LIN {X 0,Y 97.887,Z 1237.383,A -85,B 0,C 180,E1 6299.415,E2 6299.415} C_VEL
LIN {X 0,Y 98.034,Z 1228.188,A -85,B 0,C 180,E1 6290.015,E2 6290.015} C_VEL
LIN {X 0,Y 99.742,Z 1217.391,A -85,B 0,C 180,E1 6280.681,E2 6280.681} C_VEL
LIN {X 0,Y 103.666,Z 1203.945,A -85,B 0,C 180,E1 6271.166,E2 6271.166} C_VEL
LIN {X 0,Y 109.754,Z 1188.232,A -85,B 0,C 180,E1 6262.382,E2 6262.382} C_VEL
LIN {X 0,Y 117.294,Z 1170.977,A -85,B 0,C 180,E1 6254.964,E2 6254.964} C_VEL
LIN {X 0,Y 126.05,Z 1151.43,A -85,B 0,C 180,E1 6248.615,E2 6248.615} C_VEL
LIN {X 0,Y 134.664,Z 1131.582,A -85,B 0,C 180,E1 6243.735,E2 6243.735} C_VEL
LIN {X 0,Y 143.408,Z 1109.972,A -85,B 0,C 180,E1 6239.678,E2 6239.678} C_VEL
LIN {X 0,Y 151.809,Z 1086.999,A -85,B 0,C 180,E1 6236.392,E2 6236.392} C_VEL
LIN {X 0,Y 159.531,Z 1062.769,A -85,B 0,C 180,E1 6233.781,E2 6233.781} C_VEL
LIN {X 0,Y 166.358,Z 1037.239,A -85,B 0,C 180,E1 6231.721,E2 6231.721} C_VEL
LIN {X 0,Y 172.936,Z 1006.828,A -85,B 0,C 180,E1 6229.946,E2 6229.946} C_VEL
LIN {X 0,Y 199.574,Z 875.262,A -85,B 0,C 180,E1 6223.956,E2 6223.956} C_VEL
LIN {X 0,Y 191.929,Z 857.117,A -85,B 0,C 180,E1 6219.336,E2 6219.336} C_VEL
LIN {X 0,Y 189.274,Z 851.106,A -85,B 0,C 180,E1 6217.593,E2 6217.593} C_VEL
LIN {X 0,Y 178.803,Z 851.706,A -85,B 0,C 180,E1 6213.21,E2 6213.21} C_VEL
LIN {X 0,Y 172.646,Z 852.687,A -85,B 0,C 180,E1 6210.336,E2 6210.336} C_VEL
LIN {X 0,Y 172.301,Z 852.796,A -85,B 0,C 180,E1 6210.005,E2 6210.005} C_VEL
LIN {X 0,Y 174.367,Z 862.241,A -85,B 0,C 180,E1 6204.74,E2 6204.74} C_VEL
LIN {X 0,Y 176.288,Z 872.484,A -85,B 0,C 180,E1 6199.878,E2 6199.878} C_VEL
LIN {X 0,Y 177.364,Z 878.928,A -85,B 0,C 180,E1 6197.138,E2 6197.138} C_VEL
LIN {X 0,Y 158.759,Z 919.889,A -85,B 0,C 180,E1 6190.392,E2 6190.392} C_VEL
LIN {X 0,Y 148.341,Z 945.278,A -85,B 0,C 180,E1 6185.723,E2 6185.723} C_VEL
LIN {X 0,Y 137.778,Z 997.668,A -85,B 0,C 180,E1 6181.773,E2 6181.773} C_VEL
LIN {X 0,Y 129.127,Z 1037.304,A -85,B 0,C 180,E1 6177.711,E2 6177.711} C_VEL
LIN {X 0,Y 121.131,Z 1075.16,A -85,B 0,C 180,E1 6172.359,E2 6172.359} C_VEL
LIN {X 0,Y 114.899,Z 1104.872,A -85,B 0,C 180,E1 6166.97,E2 6166.97} C_VEL
LIN {X 0,Y 110.727,Z 1122.822,A -85,B 0,C 180,E1 6162.631,E2 6162.631} C_VEL
LIN {X 0,Y 106.388,Z 1140.626,A -85,B 0,C 180,E1 6156.978,E2 6156.978} C_VEL
LIN {X 0,Y 102.602,Z 1157.03,A -85,B 0,C 180,E1 6150.125,E2 6150.125} C_VEL
LIN {X 0,Y 99.911,Z 1172.201,A -85,B 0,C 180,E1 6142.043,E2 6142.043} C_VEL
LIN {X 0,Y 98.885,Z 1185.197,A -85,B 0,C 180,E1 6133.448,E2 6133.448} C_VEL
LIN {X 0,Y 99.901,Z 1197.747,A -85,B 0,C 180,E1 6123.443,E2 6123.443} C_VEL
LIN {X 0,Y 103.676,Z 1208.574,A -85,B 0,C 180,E1 6113.354,E2 6113.354} C_VEL
LIN {X 0,Y 111.219,Z 1218.395,A -85,B 0,C 180,E1 6103.28,E2 6103.28} C_VEL
LIN {X 0,Y 121.938,Z 1226.206,A -85,B 0,C 180,E1 6094.761,E2 6094.761} C_VEL
LIN {X 0,Y 135.217,Z 1232.33,A -85,B 0,C 180,E1 6087.831,E2 6087.831} C_VEL
LIN {X 0,Y 136.518,Z 1232.8,A -85,B 0,C 180,E1 6087.227,E2 6087.227} C_VEL
LIN {X 0,Y 118.677,Z 1232.303,A -85,B 0,C 180,E1 6076.965,E2 6076.965} C_VEL
LIN {X 0,Y 106.411,Z 1230.035,A -85,B 0,C 180,E1 6063.015,E2 6063.015} C_VEL
LIN {X 0,Y 102.356,Z 1226.826,A -85,B 0,C 180,E1 6049.539,E2 6049.539} C_VEL
LIN {X 0,Y 100.081,Z 1234.32,A -85,B 0,C 180,E1 6042.689,E2 6042.689} C_VEL
LIN {X 0,Y 100.4,Z 1243.403,A -85,B 0,C 180,E1 6033.418,E2 6033.418} C_VEL
LIN {X 0,Y 101.103,Z 1248.402,A -85,B 0,C 180,E1 6027.289,E2 6027.289} C_VEL
LIN {X 0,Y 100.503,Z 1252.479,A -85,B 0,C 180,E1 6020.255,E2 6020.255} C_VEL
LIN {X 0,Y 101.871,Z 1258.148,A -85,B 0,C 180,E1 6007.485,E2 6007.485} C_VEL
LIN {X 0,Y 110.666,Z 1263.588,A -85,B 0,C 180,E1 5992.084,E2 5992.084} C_VEL
LIN {X 0,Y 121.471,Z 1266.388,A -85,B 0,C 180,E1 5982.886,E2 5982.886} C_VEL
LIN {X 0,Y 107.03,Z 1258.469,A -85,B 0,C 180,E1 5969.679,E2 5969.679} C_VEL
LIN {X 0,Y 100.21,Z 1250.109,A -85,B 0,C 180,E1 5956.223,E2 5956.223} C_VEL
LIN {X 0,Y 98.516,Z 1244.153,A -85,B 0,C 180,E1 5947.728,E2 5947.728} C_VEL
LIN {X 0,Y 97.429,Z 1241.284,A -85,B 0,C 180,E1 5944.285,E2 5944.285} C_VEL
LIN {X 0,Y 94.368,Z 1236.245,A -85,B 0,C 180,E1 5939.417,E2 5939.417} C_VEL
LIN {X 0,Y 90.477,Z 1228.309,A -85,B 0,C 180,E1 5932.092,E2 5932.092} C_VEL
LIN {X 0,Y 90.289,Z 1225.819,A -85,B 0,C 180,E1 5929.68,E2 5929.68} C_VEL
LIN {X 0,Y 92.562,Z 1213.132,A -85,B 0,C 180,E1 5918.301,E2 5918.301} C_VEL
LIN {X 0,Y 97.094,Z 1199.275,A -85,B 0,C 180,E1 5908.317,E2 5908.317} C_VEL
LIN {X 0,Y 103.753,Z 1183.262,A -85,B 0,C 180,E1 5899.419,E2 5899.419} C_VEL
LIN {X 0,Y 112.036,Z 1165.199,A -85,B 0,C 180,E1 5891.822,E2 5891.822} C_VEL
LIN {X 0,Y 121.165,Z 1145.446,A -85,B 0,C 180,E1 5885.624,E2 5885.624} C_VEL
LIN {X 0,Y 130.73,Z 1123.745,A -85,B 0,C 180,E1 5880.567,E2 5880.567} C_VEL
LIN {X 0,Y 139.834,Z 1101.198,A -85,B 0,C 180,E1 5876.642,E2 5876.642} C_VEL
LIN {X 0,Y 148.357,Z 1077.435,A -85,B 0,C 180,E1 5873.564,E2 5873.564} C_VEL
LIN {X 0,Y 155.994,Z 1052.618,A -85,B 0,C 180,E1 5871.151,E2 5871.151} C_VEL
LIN {X 0,Y 162.641,Z 1026.529,A -85,B 0,C 180,E1 5869.284,E2 5869.284} C_VEL
LIN {X 0,Y 193.734,Z 878.17,A -85,B 0,C 180,E1 5862.357,E2 5862.357} C_VEL
LIN {X 0,Y 186.305,Z 860.101,A -85,B 0,C 180,E1 5857.521,E2 5857.521} C_VEL
LIN {X 0,Y 185.651,Z 858.939,A -85,B 0,C 180,E1 5857.12,E2 5857.12} C_VEL
LIN {X 0,Y 176.249,Z 859.718,A -85,B 0,C 180,E1 5853.157,E2 5853.157} C_VEL
LIN {X 0,Y 170.537,Z 860.793,A -85,B 0,C 180,E1 5850.508,E2 5850.508} C_VEL
LIN {X 0,Y 167.56,Z 861.237,A -85,B 0,C 180,E1 5848.979,E2 5848.979} C_VEL
LIN {X 0,Y 169.349,Z 870.632,A -85,B 0,C 180,E1 5843.904,E2 5843.904} C_VEL
LIN {X 0,Y 171.097,Z 881.699,A -85,B 0,C 180,E1 5838.784,E2 5838.784} C_VEL
LIN {X 0,Y 151.835,Z 922.807,A -85,B 0,C 180,E1 5831.976,E2 5831.976} C_VEL
LIN {X 0,Y 141.907,Z 946.064,A -85,B 0,C 180,E1 5827.636,E2 5827.636} C_VEL
LIN {X 0,Y 131.769,Z 994.942,A -85,B 0,C 180,E1 5823.949,E2 5823.949} C_VEL
LIN {X 0,Y 122.484,Z 1035.814,A -85,B 0,C 180,E1 5819.688,E2 5819.688} C_VEL
LIN {X 0,Y 114.221,Z 1073.153,A -85,B 0,C 180,E1 5814.264,E2 5814.264} C_VEL
LIN {X 0,Y 107.272,Z 1104.549,A -85,B 0,C 180,E1 5808.219,E2 5808.219} C_VEL
LIN {X 0,Y 102.691,Z 1123.536,A -85,B 0,C 180,E1 5803.35,E2 5803.35} C_VEL
LIN {X 0,Y 98.236,Z 1141.098,A -85,B 0,C 180,E1 5797.273,E2 5797.273} C_VEL
LIN {X 0,Y 94.303,Z 1157.899,A -85,B 0,C 180,E1 5789.625,E2 5789.625} C_VEL
LIN {X 0,Y 91.929,Z 1171.549,A -85,B 0,C 180,E1 5781.704,E2 5781.704} C_VEL
LIN {X 0,Y 91.029,Z 1185.113,A -85,B 0,C 180,E1 5772.046,E2 5772.046} C_VEL
LIN {X 0,Y 92.336,Z 1197.001,A -85,B 0,C 180,E1 5761.862,E2 5761.862} C_VEL
LIN {X 0,Y 96.65,Z 1208.083,A -85,B 0,C 180,E1 5751.073,E2 5751.073} C_VEL
LIN {X 0,Y 104.984,Z 1218.123,A -85,B 0,C 180,E1 5740.528,E2 5740.528} C_VEL
LIN {X 0,Y 117.272,Z 1226.642,A -85,B 0,C 180,E1 5731.411,E2 5731.411} C_VEL
LIN {X 0,Y 125.448,Z 1230.609,A -85,B 0,C 180,E1 5727.032,E2 5727.032} C_VEL
LIN {X 0,Y 107.068,Z 1229.03,A -85,B 0,C 180,E1 5714.449,E2 5714.449} C_VEL
LIN {X 0,Y 97.224,Z 1225.943,A -85,B 0,C 180,E1 5699.571,E2 5699.571} C_VEL
LIN {X 0,Y 95.171,Z 1223.662,A -85,B 0,C 180,E1 5690.598,E2 5690.598} C_VEL
LIN {X 0,Y 92.47,Z 1231.439,A -85,B 0,C 180,E1 5683.116,E2 5683.116} C_VEL
LIN {X 0,Y 92.869,Z 1241.238,A -85,B 0,C 180,E1 5672.46,E2 5672.46} C_VEL
LIN {X 0,Y 93.611,Z 1245.583,A -85,B 0,C 180,E1 5666.93,E2 5666.93} C_VEL
LIN {X 0,Y 93.072,Z 1249.743,A -85,B 0,C 180,E1 5659.468,E2 5659.468} C_VEL
LIN {X 0,Y 95.246,Z 1256.019,A -85,B 0,C 180,E1 5644.497,E2 5644.497} C_VEL
LIN {X 0,Y 104.166,Z 1261.116,A -85,B 0,C 180,E1 5629.965,E2 5629.965} C_VEL
LIN {X 0,Y 111.943,Z 1263.337,A -85,B 0,C 180,E1 5622.928,E2 5622.928} C_VEL
LIN {X 0,Y 98.365,Z 1255.108,A -85,B 0,C 180,E1 5609.204,E2 5609.204} C_VEL
LIN {X 0,Y 92.313,Z 1246.777,A -85,B 0,C 180,E1 5595.711,E2 5595.711} C_VEL
LIN {X 0,Y 90.586,Z 1239.38,A -85,B 0,C 180,E1 5585.066,E2 5585.066} C_VEL
LIN {X 0,Y 90.075,Z 1232.014,A -85,B 0,C 180,E1 5576.181,E2 5576.181} C_VEL
LIN {X 0,Y 90.289,Z 1225.819,A -85,B 0,C 180,E1 5569.68,E2 5569.68} C_VEL
LIN {X 0,Y 89.961,Z 1222.087,A -85,B 0,C 180,E1 5566.204,E2 5566.204} C_VEL
LIN {X 0,Y 87.947,Z 1215.287,A -85,B 0,C 180,E1 5560.649,E2 5560.649} C_VEL
LIN {X 0,Y 86.518,Z 1207.377,A -85,B 0,C 180,E1 5554.466,E2 5554.466} C_VEL
LIN {X 0,Y 87.163,Z 1203.687,A -85,B 0,C 180,E1 5551.683,E2 5551.683} C_VEL
LIN {X 0,Y 93.461,Z 1188.043,A -85,B 0,C 180,E1 5541.363,E2 5541.363} C_VEL
LIN {X 0,Y 101.58,Z 1170.681,A -85,B 0,C 180,E1 5532.79,E2 5532.79} C_VEL
LIN {X 0,Y 110.933,Z 1151.269,A -85,B 0,C 180,E1 5525.785,E2 5525.785} C_VEL
LIN {X 0,Y 120.861,Z 1129.964,A -85,B 0,C 180,E1 5520.169,E2 5520.169} C_VEL
LIN {X 0,Y 130.183,Z 1108.268,A -85,B 0,C 180,E1 5515.969,E2 5515.969} C_VEL
LIN {X 0,Y 139.174,Z 1084.923,A -85,B 0,C 180,E1 5512.602,E2 5512.602} C_VEL
LIN {X 0,Y 147.351,Z 1060.484,A -85,B 0,C 180,E1 5509.976,E2 5509.976} C_VEL
LIN {X 0,Y 154.289,Z 1035.612,A -85,B 0,C 180,E1 5508.004,E2 5508.004} C_VEL
LIN {X 0,Y 161.734,Z 1002.514,A -85,B 0,C 180,E1 5506.117,E2 5506.117} C_VEL
LIN {X 0,Y 187.811,Z 880.695,A -85,B 0,C 180,E1 5500.588,E2 5500.588} C_VEL
LIN {X 0,Y 182.236,Z 866.755,A -85,B 0,C 180,E1 5496.726,E2 5496.726} C_VEL
LIN {X 0,Y 172.721,Z 867.855,A -85,B 0,C 180,E1 5492.659,E2 5492.659} C_VEL
LIN {X 0,Y 165.989,Z 869.401,A -85,B 0,C 180,E1 5489.484,E2 5489.484} C_VEL
LIN {X 0,Y 162.942,Z 870.111,A -85,B 0,C 180,E1 5487.895,E2 5487.895} C_VEL
LIN {X 0,Y 162.827,Z 870.504,A -85,B 0,C 180,E1 5487.541,E2 5487.541} C_VEL
LIN {X 0,Y 164.415,Z 880.666,A -85,B 0,C 180,E1 5482.316,E2 5482.316} C_VEL
LIN {X 0,Y 164.929,Z 884.517,A -85,B 0,C 180,E1 5480.54,E2 5480.54} C_VEL
LIN {X 0,Y 144.85,Z 925.944,A -85,B 0,C 180,E1 5473.641,E2 5473.641} C_VEL
LIN {X 0,Y 135.621,Z 946.831,A -85,B 0,C 180,E1 5469.716,E2 5469.716} C_VEL
LIN {X 0,Y 124.493,Z 998.294,A -85,B 0,C 180,E1 5465.728,E2 5465.728} C_VEL
LIN {X 0,Y 115.046,Z 1038.311,A -85,B 0,C 180,E1 5461.381,E2 5461.381} C_VEL
LIN {X 0,Y 106.544,Z 1074.786,A -85,B 0,C 180,E1 5455.676,E2 5455.676} C_VEL
LIN {X 0,Y 99.433,Z 1105.32,A -85,B 0,C 180,E1 5449.396,E2 5449.396} C_VEL
